							IF HMI_WorkAreaDataPicking[i].NumElementiDaLavorare > 0 THEN 
								NuEstacionesPiking := NuEstacionesPiking + 1 ;	
								PosCavalleteOrdenPikin[i]	:=  e_Tipo_Pallet.CAVALLETTO;  
							END_IF
							BUNDLE_VERT:
								WorkareaState[i].Supporto.Tipologia := e_Tipo_Pallet.BUNDLE;	
							
						 ELSE
								WorkareaState[i].Supporto.Tipologia := e_Tipo_Pallet.CASSA_STANDARD;		   
						 END_CASE
					ELSE
						NumPostazioneDeposito := i; NuEstacionPiking := i;
						
						HMI_WorkAreaDataPicking[NumPostazioneDeposito].NumElementiDaLavorare := RequestPickingListFromHMI[IdxLista].SlabNumber;
						CASE HMI_WorkAreaDataPicking[i].Typology OF
							LEGNO_PIANO,TELAIO_PIANO:
								WorkareaState[i].Supporto.Tipologia := e_Tipo_Pallet.CASSA_STANDARD;
							A_FRAME_VERT:	
								WorkareaState[i].Supporto.Tipologia := e_Tipo_Pallet.CAVALLETTO;
								NuEstacionesPiking := NuEstacionesPiking + 1 ;	
								PosCavalleteOrdenPikin[i]	:=  e_Tipo_Pallet.CAVALLETTO;  	 
							BUNDLE_VERT:
								WorkareaState[i].Supporto.Tipologia := e_Tipo_Pallet.BUNDLE;	
								
							
						 ELSE
								WorkareaState[i].Supporto.Tipologia := e_Tipo_Pallet.CASSA_STANDARD;		   
						 END_CASE
					END_IF

		  
//HMI_NumeroPezziPresentiPostazione[i] := WorkAreaState[i].P -1; //NB:cancellato xckè alla attivazione azzerava il num.pezzi presenti sulle postazioni di prelievo
				END_FOR
	
				IF ElementiDaDepositare[IdxLista] <= HMI_WorkAreaDataPicking[NumPostazioneDeposito].NumElementiDaLavorare THEN
					ActualPickingListFromHMI[IdxLista] 			:= RequestPickingListFromHMI[IdxLista];
					ActualPickingListFromHMI[IdxLista].State 	:= e_StatoWorkOrder.DA_ESEGUIRE;

				ELSE
					HMI_ErroreCalcoloLista := 1;
				END_IF
				Cmd_AttivaLista[IdxLista] 				:= FALSE;
				 
			ELSE
				Cmd_AttivaLista[IdxLista] 				:= FALSE;
				 
			END_IF
{endregion}	

{region "Cotas posicione de trabajo"}

//--------------------------------------------------------------------				
//////// attivazione lista di picking : StatoWorkOrder.DA_ESEGUIRE ///
//--------------------------------------------------------------------				
			IF ActualPickingListFromHMI[IdxLista].State = e_StatoWorkOrder.DA_ESEGUIRE  THEN
				ListaInEsecuzione[IdxLista] := FALSE;
				NumeroListaInEsecuzione := 0;
			
				(* Inserimento sequenza di prelievo dalle postazioni in base al quello che l'operatore ha editato da HMI*)
				ElementiDaDepositare[IdxLista] := 0;
				ElementiElaborati[IdxLista]    := 1;
				NumPostazioneDeposito := 0;
				//FOR i:= 1 TO MAXAREAPRESENT DO
				//	WorkAreaState[i].P := 1;
				//END_FOR		
				
				FOR i:= Iforstart TO Iforend DO//---------- For 1 HMI_WorkAreaDataPicking[i].Destinazione 
					IF HMI_WorkAreaDataPicking[i].Destinazione THEN  //-------> Palet destino
						NumPostazioneDeposito := i;
						HMI_WorkAreaDataPicking[NumPostazioneDeposito].NumElementiDaLavorare 	:= RequestPickingListFromHMI[IdxLista].SlabNumber;
						(*CASE HMI_WorkAreaDataPicking[i].Typology OF     // case Pricipal1*)		 
						CASE HMI_WorkAreaDataPicking[NumPostazioneDeposito].Typology OF     // case Pricipal1	
							(* Se ho un legno in piano *)	 
							LEGNO_PIANO:	
								//WorkAreaState[NumPostazioneDeposito].Supporto.Code 						:= ActualPickingListFromHMI[IdxLista].SupportPianoLegno.Code; 
								WorkAreaState[NumPostazioneDeposito].Supporto.Code 						:= RequestPickingListFromHMIWorkArea[i].SupportPianoLegno.Code; 	   
								//WorkAreaState[NumPostazioneDeposito].Supporto.AltezzaDenteRitenuta 		:= ActualPickingListFromHMI[IdxLista].SupportPianoLegno.DimBaseUtile;
								WorkAreaState[NumPostazioneDeposito].Supporto.AltezzaDenteRitenuta 		:= RequestPickingListFromHMIWorkArea[i].SupportPianoLegno.DimBaseUtile;
								//WorkAreaState[NumPostazioneDeposito].Supporto.DimVertice 				:= ActualPickingListFromHMI[IdxLista].SupportPianoLegno.DimVertice;
								WorkAreaState[NumPostazioneDeposito].Supporto.DimVertice 				:= RequestPickingListFromHMIWorkArea[i].SupportPianoLegno.DimVertice;			   
								//WorkAreaState[NumPostazioneDeposito].Supporto.HMAX 						:= ActualPickingListFromHMI[IdxLista].SupportPianoLegno.HMAX;
							   	WorkAreaState[NumPostazioneDeposito].Supporto.HMAX 						:= RequestPickingListFromHMIWorkArea[i].SupportPianoLegno.HMAX;
								//WorkAreaState[NumPostazioneDeposito].Supporto.Tipologia 				:= e_Tipo_Pallet.CASSA_STANDARD;//ActualPickingListFromHMI.Support.Tipologia;
								WorkAreaState[NumPostazioneDeposito].Supporto.Tipologia 				:= e_Tipo_Pallet.CASSA_STANDARD;//ActualPickingListFromHMI.Support.Tipologia;   
								//WorkAreaState[NumPostazioneDeposito].Supporto.XDim 						:= ActualPickingListFromHMI[IdxLista].SupportPianoLegno.XDim;
								WorkAreaState[NumPostazioneDeposito].Supporto.XDim 						:= RequestPickingListFromHMIWorkArea[i].SupportPianoLegno.XDim;
								//WorkAreaState[NumPostazioneDeposito].Supporto.YDim 						:= ActualPickingListFromHMI[IdxLista].SupportPianoLegno.YDim;
								WorkAreaState[NumPostazioneDeposito].Supporto.YDim 						:= RequestPickingListFromHMIWorkArea[i].SupportPianoLegno.YDim;
								//WorkAreaState[NumPostazioneDeposito].Supporto.ZDim 						:= ActualPickingListFromHMI[IdxLista].SupportPianoLegno.ZDim;
								WorkAreaState[NumPostazioneDeposito].Supporto.ZDim 						:= RequestPickingListFromHMIWorkArea[i].SupportPianoLegno.ZDim;
								WorkAreaOffset[NumPostazioneDeposito].Y 								:= OFFSET_POSTAZIONE_LEGNO + ActualPickingListFromHMI[IdxLista].SupportPianoLegno.YDim/2;//ATTENZIONE!!! per poter lavorare in centro con i supporti pari, questa misura è la distanza tra il riscontro bundle verticale e il centro postazione PARI
								
								WorkAreaProductionList[NumPostazioneDeposito].Support 				:= WorkAreaState[NumPostazioneDeposito].Supporto;
								
								FOR j:= Iforstart TO Iforend DO
									IF NOT HMI_WorkAreaDataPicking[j].Destinazione THEN
										IF HMI_WorkAreaDataPicking[j].NumElementiDaLavorare >= 1 THEN
											ElementiDaDepositare[IdxLista] := ElementiElaborati[IdxLista] + HMI_WorkAreaDataPicking[j].NumElementiDaLavorare;
											FOR k := ElementiElaborati[IdxLista] TO ElementiDaDepositare[IdxLista]-1 DO	
												WorkAreaProductionList[NumPostazioneDeposito].PElementList[k].WA_PRELIEVO := j;
												WorkAreaProductionList[NumPostazioneDeposito].PElementList[k].WA_DEPOSITO := i;	
												// Se van Añadiendo los Diferentes Espesores de la receta del piking ######################################
												HMi_DimensionesPiezasWorkAreaDeposito[K] := RequestPickingListFromHMIWorkArea[j].SlabDimension ;
												//########################################################################################################
												ElementiElaborati[IdxLista] := ElementiElaborati[IdxLista]+1; 
											END_FOR
											CASE HMI_WorkAreaDataPicking[j].Typology OF 
												(* Se ho una cassa pianale in legno *)
												LEGNO_PIANO:
													WorkAreaState[j].Supporto.Code 					:= RequestPickingListFromHMIWorkArea[j].SupportPianoLegno.Code;
													WorkAreaState[j].Supporto.DimBaseUtile		 	:= RequestPickingListFromHMIWorkArea[j].SupportPianoLegno.DimBaseUtile;
													WorkAreaState[j].Supporto.AltezzaDenteRitenuta 	:= RequestPickingListFromHMIWorkArea[j].SupportPianoLegno.ZDim+20;
													WorkAreaState[j].Supporto.DimVertice 			:= RequestPickingListFromHMIWorkArea[j].SupportPianoLegno.DimVertice;
													WorkAreaState[j].Supporto.HMAX 					:= RequestPickingListFromHMIWorkArea[j].SupportPianoLegno.HMAX;
													WorkAreaState[j].Supporto.Tipologia 			:= e_Tipo_Pallet.CASSA_STANDARD;//ActualPickingListFromHMI[1].Support.Tipologia;
													WorkAreaState[j].Supporto.XDim 					:= RequestPickingListFromHMIWorkArea[j].SupportPianoLegno.XDim;
													WorkAreaState[j].Supporto.YDim 					:= RequestPickingListFromHMIWorkArea[j].SupportPianoLegno.YDim;
													WorkAreaState[j].Supporto.ZDim 					:= RequestPickingListFromHMIWorkArea[j].SupportPianoLegno.ZDim;
													WorkAreaOffset[j].Y 							:= OFFSET_POSTAZIONE_LEGNO + ActualPickingListFromHMI[IdxLista].SupportPianoLegno.YDim/2;//ATTENZIONE!!! per poter lavorare in centro con i supporti pari, questa misura è la distanza tra il riscontro bundle verticale e il centro postazione PARI
													
																   
												(* Se ho una cassa pianale in ferro su supporto *)
												TELAIO_PIANO:
													WorkAreaState[j].Supporto.Code 					:= RequestPickingListFromHMIWorkArea[j].SupportPianoFerro.Code;
													WorkAreaState[j].Supporto.DimBaseUtile		 	:= RequestPickingListFromHMIWorkArea[j].SupportPianoFerro.DimBaseUtile;
													WorkAreaState[j].Supporto.AltezzaDenteRitenuta 	:= RequestPickingListFromHMIWorkArea[j].SupportPianoFerro.ZDim+20;
													WorkAreaState[j].Supporto.DimVertice 			:= RequestPickingListFromHMIWorkArea[j].SupportPianoFerro.DimVertice;
													WorkAreaState[j].Supporto.HMAX 					:= RequestPickingListFromHMIWorkArea[j].SupportPianoFerro.HMAX;
													WorkAreaState[j].Supporto.Tipologia 			:=  e_Tipo_Pallet.CASSA_STANDARD;//ActualPickingListFromHMI[1].Support.Tipologia;
													WorkAreaState[j].Supporto.XDim 					:= RequestPickingListFromHMIWorkArea[j].SupportPianoFerro.XDim;
													WorkAreaState[j].Supporto.YDim 					:= RequestPickingListFromHMIWorkArea[j].SupportPianoFerro.YDim;
													WorkAreaState[j].Supporto.ZDim 					:= RequestPickingListFromHMIWorkArea[j].SupportPianoFerro.ZDim;
													WorkAreaOffset[j].Y 							:= OFFSET_POSTAZIONE_TELAIO - ActualPickingListFromHMI[IdxLista].SupportPianoFerro.YDim/2;//ATTENZIONE!!! per poter lavorare in centro con i supporti pari, questa misura è la distanza tra il riscontro bundle verticale e il centro postazione PARI
												(* Se ho un bundle *)
												BUNDLE_VERT:
													//WorkAreaState[j].P := ElementiDaDepositare;
													WorkAreaState[j].Supporto.Code 					:= RequestPickingListFromHMIWorkArea[j].SupportVertBundle.Code;
													WorkAreaState[j].Supporto.DimBaseUtile		 	:= RequestPickingListFromHMIWorkArea[j].SupportVertBundle.DimBaseUtile;
													WorkAreaState[j].Supporto.AltezzaDenteRitenuta 	:= RequestPickingListFromHMIWorkArea[j].SupportVertBundle.ZDim+20;
													WorkAreaState[j].Supporto.DimVertice 			:= RequestPickingListFromHMIWorkArea[j].SupportVertBundle.DimVertice;
													WorkAreaState[j].Supporto.HMAX 					:= RequestPickingListFromHMIWorkArea[j].SupportVertBundle.HMAX;
													WorkAreaState[j].Supporto.Tipologia 			:= e_Tipo_Pallet.BUNDLE;//ActualPickingListFromHMI.SupportVert.Tipologia;
													WorkAreaState[j].Supporto.XDim 					:= RequestPickingListFromHMIWorkArea[j].SupportVertBundle.XDim;
													WorkAreaState[j].Supporto.YDim 					:= RequestPickingListFromHMIWorkArea[j].SupportVertBundle.YDim;
													WorkAreaState[j].Supporto.ZDim 					:= RequestPickingListFromHMIWorkArea[j].SupportVertBundle.ZDim;
													WorkAreaState[j].Supporto.ZDim_Ext1        		:= WorkAreaState[j].Supporto.ZDim + 20;
													WorkAreaState[j].Supporto.TipoPianoAppoggio 	:= 1;                      
													WorkAreaState[j].Supporto.AltezzaDenteRitenuta	:= 20; 
													WorkAreaState[j].Supporto.LatoDeposito 			:= 180;    
													//Lo que HABIA	
													//WorkAreaOffset[j].Y 							:= HMI_OffsetDepositoLastra.Y180 ;
													//Mod 25/&/2025	  
													WorkAreaOffset[NumPostazioneDeposito].Y 		:= RequestPickingListFromHMIWorkArea[j].SupportVertBundle.YDim - RequestPickingListFromHMIWorkArea[j].SupportVertBundle.DimBaseUtile -40 ;			
												(* Se ho un A_Frame *)	  
												A_FRAME_VERT:  						
													//WorkAreaState[j].P := ElementiDaDepositare;
													WorkAreaState[j].Supporto.Code 					:= ActualPickingListFromHMI[IdxLista].SupportVertCav.Code;
													WorkAreaState[j].Supporto.DimBaseUtile		 	:= RequestPickingListFromHMIWorkArea[j].SupportVertCav.DimBaseUtile;
													WorkAreaState[j].Supporto.AltezzaDenteRitenuta 	:= RequestPickingListFromHMIWorkArea[j].SupportVertCav.ZDim+20;
													WorkAreaState[j].Supporto.DimVertice 			:= RequestPickingListFromHMIWorkArea[j].SupportVertCav.DimVertice;
													WorkAreaState[j].Supporto.HMAX 					:= RequestPickingListFromHMIWorkArea[j].SupportVertCav.HMAX;
													WorkAreaState[j].Supporto.Tipologia 			:= CAVALLETTO;//ActualPickingListFromHMI.SupportVertCav.Tipologia;
													WorkAreaState[j].Supporto.XDim 					:= RequestPickingListFromHMIWorkArea[j].SupportVertCav.XDim;
													WorkAreaState[j].Supporto.YDim 					:= RequestPickingListFromHMIWorkArea[j].SupportVertCav.YDim;
													WorkAreaState[j].Supporto.ZDim 					:= RequestPickingListFromHMIWorkArea[j].SupportVertCav.ZDim;
													WorkAreaState[j].Supporto.ZDim_Ext1        		:= WorkAreaState[j].Supporto.ZDim + 20;	
													WorkAreaState[j].Supporto.TipoPianoAppoggio 	:= 1;                      
													WorkAreaState[j].Supporto.AltezzaDenteRitenuta	:= 15;     	
													WorkAreaOffset[j].Y 							:= OFFSET_POSTAZIONE_LEGNO + ActualPickingListFromHMI[IdxLista].SupportVertCav.YDim/2;//ATTENZIONE!!! per poter lavorare in centro con i supporti pari, questa misura è la distanza tra il riscontro bundle verticale e il centro postazione PARI
											   		CoordenadaPasillo0_Y 							:= WorkArea[j].Y +  WorkAreaOffset[j].Y  - Dimensioni_Pinza.Spessore - INGOMBRO_RISCONTRO_BUNDLE - WorkAreaState[j].Supporto.YDim /2 ;
													CoordenadaPasillo180_Y 							:= WorkArea[j].Y + WorkAreaState[j].Supporto.YDim /2 + WorkAreaOffset[j].Y  + Dimensioni_Pinza.Spessore + INGOMBRO_RISCONTRO_FRAME  ;	
											END_CASE	
											WorkAreaProductionList[j].Support := WorkAreaState[j].Supporto; 
										END_IF
									END_IF     
									TFClearApprendimento(ADR(WorkAreaState[j].Apprendimento));//Azzeramento apprendimento 
								END_FOR
								EXIT; 
							(* Se ho un telaio in piano *)	 
							TELAIO_PIANO:	
								WorkAreaState[NumPostazioneDeposito].Supporto.Code 						:= ActualPickingListFromHMI[IdxLista].SupportPianoFerro.Code;
								WorkAreaState[NumPostazioneDeposito].Supporto.AltezzaDenteRitenuta 		:= RequestPickingListFromHMIWorkArea[j].SupportPianoFerro.DimBaseUtile;
								WorkAreaState[NumPostazioneDeposito].Supporto.DimVertice 				:= RequestPickingListFromHMIWorkArea[j].SupportPianoFerro.DimVertice;
								WorkAreaState[NumPostazioneDeposito].Supporto.HMAX 						:= RequestPickingListFromHMIWorkArea[j].SupportPianoFerro.HMAX;
								WorkAreaState[NumPostazioneDeposito].Supporto.Tipologia 				:= CASSA_STANDARD;//ActualPickingListFromHMI.Support.Tipologia;
								WorkAreaState[NumPostazioneDeposito].Supporto.XDim 						:= RequestPickingListFromHMIWorkArea[j].SupportPianoFerro.XDim;
								WorkAreaState[NumPostazioneDeposito].Supporto.YDim 						:= RequestPickingListFromHMIWorkArea[j].SupportPianoFerro.YDim;
								WorkAreaState[NumPostazioneDeposito].Supporto.ZDim 						:= RequestPickingListFromHMIWorkArea[j].SupportPianoFerro.ZDim;
								WorkAreaOffset[NumPostazioneDeposito].Y 								:= OFFSET_POSTAZIONE_TELAIO - ActualPickingListFromHMI[IdxLista].SupportPianoFerro.YDim/2;//ATTENZIONE!!! per poter lavorare in centro con i supporti pari, questa misura è la distanza tra il riscontro bundle verticale e il centro postazione PARI
								
								WorkAreaProductionList[NumPostazioneDeposito].Support := WorkAreaState[NumPostazioneDeposito].Supporto;
							
								
								FOR j:= Iforstart TO Iforend DO
									IF NOT HMI_WorkAreaDataPicking[j].Destinazione THEN
										IF HMI_WorkAreaDataPicking[j].NumElementiDaLavorare >= 1 THEN
											ElementiDaDepositare[IdxLista] := ElementiElaborati[IdxLista] + HMI_WorkAreaDataPicking[j].NumElementiDaLavorare;
											FOR k := ElementiElaborati[IdxLista] TO ElementiDaDepositare[IdxLista]-1 DO	
												WorkAreaProductionList[NumPostazioneDeposito].PElementList[k].WA_PRELIEVO := j;
												WorkAreaProductionList[NumPostazioneDeposito].PElementList[k].WA_DEPOSITO := i;	
												// Se van Añadiendo los Diferentes Espesores de la receta del piking ######################################
												HMi_DimensionesPiezasWorkAreaDeposito[K] := RequestPickingListFromHMIWorkArea[j].SlabDimension ;
												//########################################################################################################
												ElementiElaborati[IdxLista] := ElementiElaborati[IdxLista]+1; 
											END_FOR
											CASE HMI_WorkAreaDataPicking[j].Typology OF 
												(* Se ho una cassa pianale in legno *)
												LEGNO_PIANO:
													WorkAreaState[j].Supporto.Code 					:= ActualPickingListFromHMI[IdxLista].SupportPianoLegno.Code;
													WorkAreaState[j].Supporto.DimBaseUtile		 	:= RequestPickingListFromHMIWorkArea[j].SupportPianoLegno.DimBaseUtile;
													WorkAreaState[j].Supporto.AltezzaDenteRitenuta 	:= RequestPickingListFromHMIWorkArea[j].SupportPianoLegno.ZDim+20;
													WorkAreaState[j].Supporto.DimVertice 			:= RequestPickingListFromHMIWorkArea[j].SupportPianoLegno.DimVertice;
													WorkAreaState[j].Supporto.HMAX 					:= RequestPickingListFromHMIWorkArea[j].SupportPianoLegno.HMAX;
													WorkAreaState[j].Supporto.Tipologia 			:=  e_Tipo_Pallet.CASSA_STANDARD;//ActualPickingListFromHMI[1].Support.Tipologia;
													WorkAreaState[j].Supporto.XDim 					:= RequestPickingListFromHMIWorkArea[j].SupportPianoLegno.XDim;
													WorkAreaState[j].Supporto.YDim 					:= RequestPickingListFromHMIWorkArea[j].SupportPianoLegno.YDim;
													WorkAreaState[j].Supporto.ZDim 					:= RequestPickingListFromHMIWorkArea[j].SupportPianoLegno.ZDim;
													WorkAreaOffset[j].Y 							:= OFFSET_POSTAZIONE_LEGNO + ActualPickingListFromHMI[IdxLista].SupportPianoLegno.YDim/2;//ATTENZIONE!!! per poter lavorare in centro con i supporti pari, questa misura è la distanza tra il riscontro bundle verticale e il centro postazione PARI
												(* Se ho una cassa pianale in ferro su supporto *)
												TELAIO_PIANO:
													WorkAreaState[j].Supporto.Code 					:= ActualPickingListFromHMI[IdxLista].SupportPianoFerro.Code;
													WorkAreaState[j].Supporto.DimBaseUtile		 	:= RequestPickingListFromHMIWorkArea[j].SupportPianoFerro.DimBaseUtile;
													WorkAreaState[j].Supporto.AltezzaDenteRitenuta 	:= RequestPickingListFromHMIWorkArea[j].SupportPianoFerro.ZDim+20;
													WorkAreaState[j].Supporto.DimVertice 			:= RequestPickingListFromHMIWorkArea[j].SupportPianoFerro.DimVertice;
													WorkAreaState[j].Supporto.HMAX 					:= RequestPickingListFromHMIWorkArea[j].SupportPianoFerro.HMAX;
													WorkAreaState[j].Supporto.Tipologia 			:=  e_Tipo_Pallet.CASSA_STANDARD;//ActualPickingListFromHMI[1].Support.Tipologia;
													WorkAreaState[j].Supporto.XDim 					:= RequestPickingListFromHMIWorkArea[j].SupportPianoFerro.XDim;
													WorkAreaState[j].Supporto.YDim 					:= RequestPickingListFromHMIWorkArea[j].SupportPianoFerro.YDim;
													WorkAreaState[j].Supporto.ZDim 					:= RequestPickingListFromHMIWorkArea[j].SupportPianoFerro.ZDim;
													WorkAreaOffset[j].Y 							:= OFFSET_POSTAZIONE_TELAIO - ActualPickingListFromHMI[IdxLista].SupportPianoFerro.YDim/2;//ATTENZIONE!!! per poter lavorare in centro con i supporti pari, questa misura è la distanza tra il riscontro bundle verticale e il centro postazione PARI
												(* Se ho un bundle *)
												BUNDLE_VERT:
													//WorkAreaState[j].P := ElementiDaDepositare;
													WorkAreaState[j].Supporto.Code 					:= RequestPickingListFromHMIWorkArea[j].SupportVertBundle.Code;
													WorkAreaState[j].Supporto.DimBaseUtile		 	:= RequestPickingListFromHMIWorkArea[j].SupportVertBundle.DimBaseUtile;
													WorkAreaState[j].Supporto.AltezzaDenteRitenuta 	:= RequestPickingListFromHMIWorkArea[j].SupportVertBundle.ZDim+20;
													WorkAreaState[j].Supporto.DimVertice 			:= RequestPickingListFromHMIWorkArea[j].SupportVertBundle.DimVertice;
													WorkAreaState[j].Supporto.HMAX 					:= RequestPickingListFromHMIWorkArea[j].SupportVertBundle.HMAX;
													WorkAreaState[j].Supporto.Tipologia 			:= e_Tipo_Pallet.BUNDLE;//ActualPickingListFromHMI.SupportVertBundle.Tipologia;
													WorkAreaState[j].Supporto.XDim 					:= RequestPickingListFromHMIWorkArea[j].SupportVertBundle.XDim;
													WorkAreaState[j].Supporto.YDim 					:= RequestPickingListFromHMIWorkArea[j].SupportVertBundle.YDim;
													WorkAreaState[j].Supporto.ZDim 					:= RequestPickingListFromHMIWorkArea[j].SupportVertBundle.ZDim;
													WorkAreaState[j].Supporto.ZDim_Ext1        		:= WorkAreaState[j].Supporto.ZDim + 20;
													WorkAreaState[j].Supporto.TipoPianoAppoggio 	:= 1;                      
													WorkAreaState[j].Supporto.AltezzaDenteRitenuta	:= 20; 
													WorkAreaState[j].Supporto.LatoDeposito 			:= 180;   	
													  
													WorkAreaOffset[j].Y 		:= 0 ;	
													//Mod 25/&/2025	  
													//WorkAreaOffset[j].Y 		:= ActualPickingListFromHMI[IdxLista].SupportVertBundle.YDim-ActualPickingListFromHMI[IdxLista].SupportVertBundle.DimBaseUtile -40;				
												(* Se ho un A_Frame *)	  
												A_FRAME_VERT:  						
													//WorkAreaState[j].P := ElementiDaDepositare;
													WorkAreaState[j].Supporto.Code 					:= ActualPickingListFromHMI[IdxLista].SupportVertCav.Code;
													WorkAreaState[j].Supporto.DimBaseUtile		 	:= RequestPickingListFromHMIWorkArea[j].SupportVertCav.DimBaseUtile;
													WorkAreaState[j].Supporto.AltezzaDenteRitenuta 	:= RequestPickingListFromHMIWorkArea[j].SupportVertCav.ZDim+20;
													WorkAreaState[j].Supporto.DimVertice 			:= RequestPickingListFromHMIWorkArea[j].SupportVertCav.DimVertice;
													WorkAreaState[j].Supporto.HMAX 					:= RequestPickingListFromHMIWorkArea[j].SupportVertcav.HMAX;
													WorkAreaState[j].Supporto.Tipologia 			:= CAVALLETTO;//ActualPickingListFromHMI.SupportVert.Tipologia;
													WorkAreaState[j].Supporto.XDim 					:= RequestPickingListFromHMIWorkArea[j].SupportVertCav.XDim;
													WorkAreaState[j].Supporto.YDim 					:= RequestPickingListFromHMIWorkArea[j].SupportVertCav.YDim;
													WorkAreaState[j].Supporto.ZDim 					:= RequestPickingListFromHMIWorkArea[j].SupportVertCav.ZDim;
													WorkAreaState[j].Supporto.ZDim_Ext1        		:= WorkAreaState[j].Supporto.ZDim + 20;	
													WorkAreaState[j].Supporto.TipoPianoAppoggio 	:= 1;                      
													WorkAreaState[j].Supporto.AltezzaDenteRitenuta	:= 15; 	
													WorkAreaOffset[j].Y 							:= OFFSET_POSTAZIONE_LEGNO + ActualPickingListFromHMI[IdxLista].SupportVertCav.YDim/2;//ATTENZIONE!!! per poter lavorare in centro con i supporti pari, questa misura è la distanza tra il riscontro bundle verticale e il centro postazione PARI
											   		CoordenadaPasillo0_Y 							:= WorkArea[j].Y +  WorkAreaOffset[j].Y  - Dimensioni_Pinza.Spessore - INGOMBRO_RISCONTRO_BUNDLE - WorkAreaState[j].Supporto.YDim /2 ;
													CoordenadaPasillo180_Y 							:= WorkArea[j].Y + WorkAreaState[j].Supporto.YDim /2 + WorkAreaOffset[j].Y  + Dimensioni_Pinza.Spessore + INGOMBRO_RISCONTRO_FRAME  ;	
											END_CASE	
											WorkAreaProductionList[j].Support := WorkAreaState[j].Supporto; 
										END_IF
									END_IF     
									TFClearApprendimento(ADR(WorkAreaState[j].Apprendimento));//Azzeramento apprendimento 
								END_FOR
								EXIT; 
							(* Se ho un bundle *)
							BUNDLE_VERT:
								
								//Se ho deposito verticale su bundle
								WorkAreaState[NumPostazioneDeposito].Supporto.Code 						:= ActualPickingListFromHMI[IdxLista].SupportVertBundle.Code;
								WorkAreaState[NumPostazioneDeposito].Supporto.DimBaseUtile		 		:= RequestPickingListFromHMIWorkArea[j].SupportVertBundle.DimBaseUtile;
								WorkAreaState[NumPostazioneDeposito].Supporto.DimVertice 				:= RequestPickingListFromHMIWorkArea[j].SupportVertBundle.DimVertice;
								WorkAreaState[NumPostazioneDeposito].Supporto.HMAX 						:= RequestPickingListFromHMIWorkArea[j].SupportVertBundle.HMAX;
								WorkAreaState[NumPostazioneDeposito].Supporto.Tipologia 				:= e_Tipo_Pallet.BUNDLE;
								WorkAreaState[NumPostazioneDeposito].Supporto.XDim 						:= RequestPickingListFromHMIWorkArea[j].SupportVertBundle.XDim;
								WorkAreaState[NumPostazioneDeposito].Supporto.YDim 						:= RequestPickingListFromHMIWorkArea[j].SupportVertBundle.YDim;
								WorkAreaState[NumPostazioneDeposito].Supporto.ZDim 						:= RequestPickingListFromHMIWorkArea[j].SupportVertBundle.ZDim;
								WorkAreaState[NumPostazioneDeposito].Supporto.TipoPianoAppoggio 		:= 1;                      
								WorkAreaState[NumPostazioneDeposito].Supporto.AltezzaDenteRitenuta		:= 20; 
								WorkAreaState[NumPostazioneDeposito].Supporto.LatoDeposito 				:= 180; 
											   
								WorkAreaProductionList[NumPostazioneDeposito].Support 					:= WorkAreaState[NumPostazioneDeposito].Supporto;
								
								FOR j:= Iforstart TO Iforend DO
									IF NOT HMI_WorkAreaDataPicking[j].Destinazione THEN
										IF HMI_WorkAreaDataPicking[j].NumElementiDaLavorare >= 1 THEN
											ElementiDaDepositare[IdxLista] := ElementiElaborati[IdxLista] + HMI_WorkAreaDataPicking[j].NumElementiDaLavorare;
											FOR k := ElementiElaborati[IdxLista] TO ElementiDaDepositare[IdxLista]-1 DO	
												WorkAreaProductionList[NumPostazioneDeposito].PElementList[k].WA_PRELIEVO := j;
												WorkAreaProductionList[NumPostazioneDeposito].PElementList[k].WA_DEPOSITO := i;	
												// Se van Añadiendo los Diferentes Espesores de la receta del piking ######################################
												HMi_DimensionesPiezasWorkAreaDeposito[K] := RequestPickingListFromHMIWorkArea[j].SlabDimension ;
												//########################################################################################################
												ElementiElaborati[IdxLista] := ElementiElaborati[IdxLista]+1; 
											END_FOR
											CASE HMI_WorkAreaDataPicking[j].Typology OF 
												(* Se ho una cassa pianale in legno *)
												LEGNO_PIANO:
													WorkAreaState[j].Supporto.Code 					:= ActualPickingListFromHMI[IdxLista].SupportPianoLegno.Code;
													WorkAreaState[j].Supporto.DimBaseUtile		 	:= RequestPickingListFromHMIWorkArea[j].SupportPianoLegno.DimBaseUtile;
													WorkAreaState[j].Supporto.AltezzaDenteRitenuta 	:= RequestPickingListFromHMIWorkArea[j].SupportPianoLegno.ZDim+20;
													WorkAreaState[j].Supporto.DimVertice 			:= RequestPickingListFromHMIWorkArea[j].SupportPianoLegno.DimVertice;
													WorkAreaState[j].Supporto.HMAX 					:= RequestPickingListFromHMIWorkArea[j].SupportPianoLegno.HMAX;
													WorkAreaState[j].Supporto.Tipologia 			:=  e_Tipo_Pallet.CASSA_STANDARD;//ActualPickingListFromHMI[1].Support.Tipologia;
													WorkAreaState[j].Supporto.XDim 					:= RequestPickingListFromHMIWorkArea[j].SupportPianoLegno.XDim;
													WorkAreaState[j].Supporto.YDim 					:= RequestPickingListFromHMIWorkArea[j].SupportPianoLegno.YDim;
													WorkAreaState[j].Supporto.ZDim 					:= RequestPickingListFromHMIWorkArea[j].SupportPianoLegno.ZDim;
													WorkAreaOffset[j].Y 							:= OFFSET_POSTAZIONE_LEGNO + ActualPickingListFromHMI[IdxLista].SupportPianoLegno.YDim/2;//ATTENZIONE!!! per poter lavorare in centro con i supporti pari, questa misura è la distanza tra il riscontro bundle verticale e il centro postazione PARI
												(* Se ho una cassa pianale in ferro su supporto *)
												TELAIO_PIANO:
													WorkAreaState[j].Supporto.Code 					:= ActualPickingListFromHMI[IdxLista].SupportPianoFerro.Code;
													WorkAreaState[j].Supporto.DimBaseUtile		 	:= RequestPickingListFromHMIWorkArea[j].SupportPianoFerro.DimBaseUtile;
													WorkAreaState[j].Supporto.AltezzaDenteRitenuta 	:= RequestPickingListFromHMIWorkArea[j].SupportPianoFerro.ZDim+20;
													WorkAreaState[j].Supporto.DimVertice 			:= RequestPickingListFromHMIWorkArea[j].SupportPianoFerro.DimVertice;
													WorkAreaState[j].Supporto.HMAX 					:= RequestPickingListFromHMIWorkArea[j].SupportPianoFerro.HMAX;
													WorkAreaState[j].Supporto.Tipologia 			:=  e_Tipo_Pallet.CASSA_STANDARD;//ActualPickingListFromHMI[1].Support.Tipologia;
													WorkAreaState[j].Supporto.XDim 					:= RequestPickingListFromHMIWorkArea[j].SupportPianoFerro.XDim;
													WorkAreaState[j].Supporto.YDim 					:= RequestPickingListFromHMIWorkArea[j].SupportPianoFerro.YDim;
													WorkAreaState[j].Supporto.ZDim 					:= RequestPickingListFromHMIWorkArea[j].SupportPianoFerro.ZDim;
													WorkAreaOffset[j].Y 							:= OFFSET_POSTAZIONE_TELAIO - ActualPickingListFromHMI[IdxLista].SupportPianoFerro.YDim/2;//ATTENZIONE!!! per poter lavorare in centro con i supporti pari, questa misura è la distanza tra il riscontro bundle verticale e il centro postazione PARI
												(* Se ho un bundle *)
												BUNDLE_VERT:
													//WorkAreaState[j].P := ElementiDaDepositare;
													WorkAreaState[j].Supporto.Code 					:= ActualPickingListFromHMI[IdxLista].SupportVertBundle.Code;
													WorkAreaState[j].Supporto.DimBaseUtile		 	:= RequestPickingListFromHMIWorkArea[j].SupportVertBundle.DimBaseUtile;
													WorkAreaState[j].Supporto.AltezzaDenteRitenuta 	:= RequestPickingListFromHMIWorkArea[j].SupportVertBundle.ZDim+20;
													WorkAreaState[j].Supporto.DimVertice 			:= RequestPickingListFromHMIWorkArea[j].SupportVertBundle.DimVertice;
													WorkAreaState[j].Supporto.HMAX 					:= RequestPickingListFromHMIWorkArea[j].SupportVertBundle.HMAX;
													WorkAreaState[j].Supporto.Tipologia 			:= e_Tipo_Pallet.BUNDLE;//ActualPickingListFromHMI.SupportVert.Tipologia;
													WorkAreaState[j].Supporto.XDim 					:= RequestPickingListFromHMIWorkArea[j].SupportVertBundle.XDim;
													WorkAreaState[j].Supporto.YDim 					:= RequestPickingListFromHMIWorkArea[j].SupportVertBundle.YDim;
													WorkAreaState[j].Supporto.ZDim 					:= RequestPickingListFromHMIWorkArea[j].SupportVertBundle.ZDim;
													WorkAreaState[j].Supporto.ZDim_Ext1        		:= WorkAreaState[j].Supporto.ZDim + 20;	
													// **Lo Que Habia	
													WorkAreaOffset[j].Y 							:= 0;
													//Mod 25/&/2025	  
													//WorkAreaOffset[j].Y 		:= ActualPickingListFromHMI[IdxLista].SupportVertBundle.YDim-ActualPickingListFromHMI[IdxLista].SupportVertBundle.DimBaseUtile -40;	
			
												(* Se ho un A_Frame *)	  
												A_FRAME_VERT:  						
													//WorkAreaState[j].P := ElementiDaDepositare;
													WorkAreaState[j].Supporto.Code 					:= ActualPickingListFromHMI[IdxLista].SupportVertCav.Code;
													WorkAreaState[j].Supporto.DimBaseUtile		 	:= RequestPickingListFromHMIWorkArea[j].SupportVertCav.DimBaseUtile;
													WorkAreaState[j].Supporto.AltezzaDenteRitenuta 	:= RequestPickingListFromHMIWorkArea[j].SupportVertCav.ZDim+20;
													WorkAreaState[j].Supporto.DimVertice 			:= RequestPickingListFromHMIWorkArea[j].SupportVertCav.DimVertice;
													WorkAreaState[j].Supporto.HMAX 					:= RequestPickingListFromHMIWorkArea[j].SupportVertCav.HMAX;
													WorkAreaState[j].Supporto.Tipologia 			:= CAVALLETTO;//ActualPickingListFromHMI.SupportVert.Tipologia;
													WorkAreaState[j].Supporto.XDim 					:= RequestPickingListFromHMIWorkArea[j].SupportVertCav.XDim;
													WorkAreaState[j].Supporto.YDim 					:= RequestPickingListFromHMIWorkArea[j].SupportVertCav.YDim;
													WorkAreaState[j].Supporto.ZDim 					:= RequestPickingListFromHMIWorkArea[j].SupportVertCav.ZDim;
													WorkAreaState[j].Supporto.ZDim_Ext1        		:= WorkAreaState[j].Supporto.ZDim + 20;	
													WorkAreaState[j].Supporto.TipoPianoAppoggio 	:= 1;                      
													WorkAreaState[j].Supporto.AltezzaDenteRitenuta	:= 15; 	
													WorkAreaOffset[j].Y 							:= OFFSET_POSTAZIONE_LEGNO + ActualPickingListFromHMI[IdxLista].SupportVertCav.YDim/2;//ATTENZIONE!!! per poter lavorare in centro con i supporti pari, questa misura è la distanza tra il riscontro bundle verticale e il centro postazione PARI
													CoordenadaPasillo0_Y 							:= WorkArea[j].Y +  WorkAreaOffset[j].Y  - Dimensioni_Pinza.Spessore - INGOMBRO_RISCONTRO_BUNDLE - WorkAreaState[j].Supporto.YDim /2 ;
													CoordenadaPasillo180_Y 							:= WorkArea[j].Y + WorkAreaState[j].Supporto.YDim /2 + WorkAreaOffset[j].Y  + Dimensioni_Pinza.Spessore + INGOMBRO_RISCONTRO_FRAME  ;		  
											END_CASE
											//WorkAreaProductionList[j].Support := HMI_Formatura.HMI_Forming_Supporto;		  
											WorkAreaProductionList[j].Support := WorkAreaState[j].Supporto;
										END_IF
									END_IF
									TFClearApprendimento(ADR(WorkAreaState[j].Apprendimento));//Azzeramento apprendimento
								END_FOR
								EXIT; 
							(* Se ho un A_Frame *)	
							A_FRAME_VERT:
								WorkAreaState[NumPostazioneDeposito].Supporto.Code 						:= ActualPickingListFromHMI[IdxLista].SupportVertCav.Code;
								WorkAreaState[NumPostazioneDeposito].Supporto.DimBaseUtile		 		:= RequestPickingListFromHMIWorkArea[j].SupportVertCav.DimBaseUtile;
								WorkAreaState[NumPostazioneDeposito].Supporto.DimVertice 				:= RequestPickingListFromHMIWorkArea[j].SupportVertCav.DimVertice;
								WorkAreaState[NumPostazioneDeposito].Supporto.HMAX 						:= RequestPickingListFromHMIWorkArea[j].SupportVertCav.HMAX;
								WorkAreaState[NumPostazioneDeposito].Supporto.Tipologia 				:= e_Tipo_Pallet.CAVALLETTO;//ActualPickingListFromHMI.SupportVertBundle.Tipologia;
								WorkAreaState[NumPostazioneDeposito].Supporto.XDim 						:= RequestPickingListFromHMIWorkArea[j].SupportVertCav.XDim;
								WorkAreaState[NumPostazioneDeposito].Supporto.YDim 						:= RequestPickingListFromHMIWorkArea[j].SupportVertCav.YDim;
								WorkAreaState[NumPostazioneDeposito].Supporto.ZDim 						:= RequestPickingListFromHMIWorkArea[j].SupportVertCav.ZDim;
								WorkAreaState[NumPostazioneDeposito].Supporto.TipoPianoAppoggio 		:= 1;                      
								WorkAreaState[NumPostazioneDeposito].Supporto.AltezzaDenteRitenuta		:= 15; 
								//WorkAreaOffset[NumPostazioneDeposito].Y 								:= OFFSET_POSTAZIONE_LEGNO (*- ActualPickingListFromHMI[IdxLista].SupportPianoFerro.YDim/2*);
								WorkAreaOffset[NumPostazioneDeposito].Y 								:= OFFSET_POSTAZIONE_LEGNO + ActualPickingListFromHMI[IdxLista].SupportVertCav.YDim/2;	
								
								WorkAreaProductionList[NumPostazioneDeposito].Support 				:= WorkAreaState[NumPostazioneDeposito].Supporto; 
								
								FOR j:= Iforstart TO Iforend DO
									IF NOT HMI_WorkAreaDataPicking[j].Destinazione THEN
										IF HMI_WorkAreaDataPicking[j].NumElementiDaLavorare >= 1 THEN
											ElementiDaDepositare[IdxLista] := ElementiElaborati[IdxLista] + HMI_WorkAreaDataPicking[j].NumElementiDaLavorare;
											FOR k := ElementiElaborati[IdxLista] TO ElementiDaDepositare[IdxLista]-1 DO	
												WorkAreaProductionList[NumPostazioneDeposito].PElementList[k].WA_PRELIEVO := j;
												WorkAreaProductionList[NumPostazioneDeposito].PElementList[k].WA_DEPOSITO := i;	
												// Se van Añadiendo los Diferentes Espesores de la receta del piking ######################################
												HMi_DimensionesPiezasWorkAreaDeposito[K] := RequestPickingListFromHMIWorkArea[j].SlabDimension ;
												//########################################################################################################
												ElementiElaborati[IdxLista] := ElementiElaborati[IdxLista]+1; 
											END_FOR
											CASE HMI_WorkAreaDataPicking[j].Typology OF 
												(* Se ho una cassa pianale in legno *)
												LEGNO_PIANO:
													WorkAreaState[j].Supporto.Code 					:= ActualPickingListFromHMI[IdxLista].SupportPianoLegno.Code;
													WorkAreaState[j].Supporto.DimBaseUtile		 	:= RequestPickingListFromHMIWorkArea[j].SupportPianoLegno.DimBaseUtile;
													WorkAreaState[j].Supporto.AltezzaDenteRitenuta 	:= RequestPickingListFromHMIWorkArea[j].SupportPianoLegno.ZDim+20;
													WorkAreaState[j].Supporto.DimVertice 			:= RequestPickingListFromHMIWorkArea[j].SupportPianoLegno.DimVertice;
													WorkAreaState[j].Supporto.HMAX 					:= RequestPickingListFromHMIWorkArea[j].SupportPianoLegno.HMAX;
													WorkAreaState[j].Supporto.Tipologia 			:=  e_Tipo_Pallet.CASSA_STANDARD;//ActualPickingListFromHMI[1].Support.Tipologia;
													WorkAreaState[j].Supporto.XDim 					:= RequestPickingListFromHMIWorkArea[j].SupportPianoLegno.XDim;
													WorkAreaState[j].Supporto.YDim 					:= RequestPickingListFromHMIWorkArea[j].SupportPianoLegno.YDim;
													WorkAreaState[j].Supporto.ZDim 					:= RequestPickingListFromHMIWorkArea[j].SupportPianoLegno.ZDim;
													WorkAreaOffset[j].Y 							:= OFFSET_POSTAZIONE_LEGNO + RequestPickingListFromHMIWorkArea[j].SupportPianoLegno.YDim/2;//ATTENZIONE!!! per poter lavorare in centro con i supporti pari, questa misura è la distanza tra il riscontro bundle verticale e il centro postazione PARI
												(* Se ho una cassa pianale in ferro su supporto *)
												TELAIO_PIANO:
													WorkAreaState[j].Supporto.Code 					:= ActualPickingListFromHMI[IdxLista].SupportPianoFerro.Code;
													WorkAreaState[j].Supporto.DimBaseUtile		 	:= RequestPickingListFromHMIWorkArea[j].SupportPianoFerro.DimBaseUtile;
													WorkAreaState[j].Supporto.AltezzaDenteRitenuta 	:= RequestPickingListFromHMIWorkArea[j].SupportPianoFerro.ZDim+20;
													WorkAreaState[j].Supporto.DimVertice 			:= RequestPickingListFromHMIWorkArea[j].SupportPianoFerro.DimVertice;
													WorkAreaState[j].Supporto.HMAX 					:= RequestPickingListFromHMIWorkArea[j].SupportPianoFerro.HMAX;
													WorkAreaState[j].Supporto.Tipologia 			:=  e_Tipo_Pallet.CASSA_STANDARD;//ActualPickingListFromHMI[1].Support.Tipologia;
													WorkAreaState[j].Supporto.XDim 					:= RequestPickingListFromHMIWorkArea[j].SupportPianoFerro.XDim;
													WorkAreaState[j].Supporto.YDim 					:= RequestPickingListFromHMIWorkArea[j].SupportPianoFerro.YDim;
													WorkAreaState[j].Supporto.ZDim 					:= RequestPickingListFromHMIWorkArea[j].SupportPianoFerro.ZDim;
													WorkAreaOffset[j].Y 							:= OFFSET_POSTAZIONE_TELAIO - RequestPickingListFromHMIWorkArea[j].SupportPianoFerro.YDim/2;//ATTENZIONE!!! per poter lavorare in centro con i supporti pari, questa misura è la distanza tra il riscontro bundle verticale e il centro postazione PARI
												(* Se ho un bundle *)
												BUNDLE_VERT:
													//WorkAreaState[j].P := ElementiDaDepositare;
													WorkAreaState[j].Supporto.Code 					:= ActualPickingListFromHMI[IdxLista].SupportVertBundle.Code;
													WorkAreaState[j].Supporto.DimBaseUtile		 	:= RequestPickingListFromHMIWorkArea[j].SupportVertBundle.DimBaseUtile;
													WorkAreaState[j].Supporto.AltezzaDenteRitenuta 	:= RequestPickingListFromHMIWorkArea[j].SupportVertBundle.ZDim+20;
													WorkAreaState[j].Supporto.DimVertice 			:= RequestPickingListFromHMIWorkArea[j].SupportVertBundle.DimVertice;
													WorkAreaState[j].Supporto.HMAX 					:= RequestPickingListFromHMIWorkArea[j].SupportVertBundle.HMAX;
													WorkAreaState[j].Supporto.Tipologia 			:= e_Tipo_Pallet.BUNDLE;//ActualPickingListFromHMI.SupportVert.Tipologia;
													WorkAreaState[j].Supporto.XDim 					:= RequestPickingListFromHMIWorkArea[j].SupportVertBundle.XDim;
													WorkAreaState[j].Supporto.YDim 					:= RequestPickingListFromHMIWorkArea[j].SupportVertBundle.YDim;
													WorkAreaState[j].Supporto.ZDim 					:= RequestPickingListFromHMIWorkArea[j].SupportVertBundle.ZDim;
													WorkAreaState[j].Supporto.ZDim_Ext1        		:= WorkAreaState[j].Supporto.ZDim + 20;	
													WorkAreaState[j].Supporto.TipoPianoAppoggio 	:= 1;                      
													WorkAreaState[j].Supporto.AltezzaDenteRitenuta	:= 20; 
													WorkAreaState[j].Supporto.LatoDeposito 			:= 180; 
													//**Lo Que Habia
													WorkAreaOffset[j].Y 							:= 0;
													//Mod 25/&/2025	  
													//WorkAreaOffset[j].Y 		:= ActualPickingListFromHMI[IdxLista].SupportVertBundle.YDim-ActualPickingListFromHMI[IdxLista].SupportVertBundle.DimBaseUtile -40;					
												(* Se ho un A_Frame *)	  
												A_FRAME_VERT:  						
													//WorkAreaState[j].P := ElementiDaDepositare;
													WorkAreaState[j].Supporto.Code 					:= ActualPickingListFromHMI[IdxLista].SupportVertCav.Code;
													WorkAreaState[j].Supporto.DimBaseUtile		 	:= RequestPickingListFromHMIWorkArea[j].SupportVertCav.DimBaseUtile;
													WorkAreaState[j].Supporto.AltezzaDenteRitenuta 	:= RequestPickingListFromHMIWorkArea[j].SupportVertCav.ZDim+20;
													WorkAreaState[j].Supporto.DimVertice 			:= RequestPickingListFromHMIWorkArea[j].SupportVertCav.DimVertice;
													WorkAreaState[j].Supporto.HMAX 					:= RequestPickingListFromHMIWorkArea[j].SupportVertCav.HMAX;
													WorkAreaState[j].Supporto.Tipologia 			:= CAVALLETTO;//ActualPickingListFromHMI.SupportVertCav.Tipologia;
													WorkAreaState[j].Supporto.XDim 					:= RequestPickingListFromHMIWorkArea[j].SupportVertCav.XDim;
													WorkAreaState[j].Supporto.YDim 					:= RequestPickingListFromHMIWorkArea[j].SupportVertCav.YDim;
													WorkAreaState[j].Supporto.ZDim 					:= RequestPickingListFromHMIWorkArea[j].SupportVertCav.ZDim;
													WorkAreaState[j].Supporto.ZDim_Ext1        		:= WorkAreaState[j].Supporto.ZDim + 20;	
													WorkAreaState[j].Supporto.TipoPianoAppoggio 	:= 1;                      
													WorkAreaState[j].Supporto.AltezzaDenteRitenuta	:= 15; 		
													WorkAreaOffset[j].Y 							:= OFFSET_POSTAZIONE_LEGNO + RequestPickingListFromHMIWorkArea[j].SupportVertCav.YDim/2;//ATTENZIONE!!! per poter lavorare in centro con i supporti pari, questa misura è la distanza tra il riscontro bundle verticale e il centro postazione PARI
												   	CoordenadaPasillo0_Y 							:= WorkArea[j].Y +  WorkAreaOffset[j].Y  - Dimensioni_Pinza.Spessore - INGOMBRO_RISCONTRO_BUNDLE - WorkAreaState[j].Supporto.YDim /2 ;
													CoordenadaPasillo180_Y 							:= WorkArea[j].Y + WorkAreaState[j].Supporto.YDim /2 + WorkAreaOffset[j].Y  + Dimensioni_Pinza.Spessore + INGOMBRO_RISCONTRO_FRAME  ;	
												
											END_CASE
													  
											WorkAreaProductionList[j].Support := WorkAreaState[j].Supporto;
										END_IF
									END_IF
									TFClearApprendimento(ADR(WorkAreaState[j].Apprendimento));//Azzeramento apprendimento
								END_FOR
								EXIT; 
						END_CASE // case Pricipal1
					END_IF	//-------->	 //-------> Palet destino
				END_FOR//----------For 1 HMI_WorkAreaDataPicking[i].Destinazione 
				
				Picking.Cmd_CalcolaLista[IdxLista] := TRUE;
				HMI_Forming_Attivazione[IdxLista] := TRUE;//attivo nuova formatura
			END_IF //------------------------------ActualPickingListFromHMI[IdxLista].State = e_StatoWorkOrder.DA_ESEGUIRE 
{endregion }
			 
		    	  


	IF Picking.Cmd_CalcolaLista[IdxLista] AND HMI_Forming_Attivazione[IdxLista] THEN
			idxForm:= IdxLista;		  
		FOR CalFor := Iforstart TO Iforend DO
				CrearFormacion := 1 ; 
				IF CalFor = NumPostazioneDeposito THEN // calcula la formacion para la estacion de piking
					CASE CrearFormacion OF
		  				1:  
							//Ack 
							IF HMI_ErrAckCalcolaFormatura THEN
								HMI_Forming_ErroreCalcoli 					:= 0;
								HMI_ErrAckCalcolaFormatura 					:= FALSE;
								FOR i:= 1 TO MAXFORMING DO
									HMI_ConfermaAttivazioneFormatura[i] 	:= FALSE;
									HMI_Forming_FormaturaAttivata[i] 		:= FALSE;
								END_FOR	 
							END_IF
							
							//Azzeramento comandi in caso di errore
							IF HMI_Forming_ErroreCalcoli <> 0 THEN
								FOR i:=1 TO MAXFORMING DO
									HMI_Forming_Attivazione[i] 				:= FALSE;
									HMI_Forming_Disattivazione[i] 			:= FALSE;
								END_FOR
								HMI_Forming_Calcola 						:= FALSE;
							END_IF
							// borra las estructuras Anteas hacer el calculo
							TFCalcoloFormaturaWA[CalFor].PulisciMemoria := TRUE ;
							HMI_Forming_FormaturaAttivata[idxForm] 		:= FALSE;	
							TFCalcoloFormaturaWA[CalFor]() ;
							CrearFormacion := 2 ; 	  
						2:
								  
							
							IF 	 TFCalcoloFormaturaWA[CalFor].PulisciMemoria AND TFCalcoloFormaturaWA[CalFor].PulisciMemoriaDone THEN 
								// borra La Formacion de la estructura		  
								WorkAreaProductionList[CalFor].Forming := FormingEmpty;
									 
								CASE WorkAreaState[NumPostazioneDeposito].Supporto.Tipologia OF //**Mod
									BUNDLE_VERT:
										TFCalcoloFormaturaWA[CalFor].TipoOrdinamento := 4;//Ordinamento di deposito òato 180°
									A_FRAME_VERT:
										TFCalcoloFormaturaWA[CalFor].TipoOrdinamento := 1;//Ordinamento di deposito, prima un lato poi l'altro	
										TFCalcoloFormaturaWA[CalFor].HabiCalTodasCordenadas := TRUE ;
									ELSE
										TFCalcoloFormaturaWA[CalFor].TipoOrdinamento := 2;//Ordinamento di deposito consecutivo	 
								END_CASE
								(*
									//Valorizzo altezza esterna supporto
									//IF HMI_Forming_Supporto.ZDim_Ext1 = 0 THEN
										HMI_Forming_Supporto.ZDim_Ext1 := HMI_Forming_Supporto.ZDim + HMI_Forming_Supporto.AltezzaDenteRitenuta;
									//END_IF
									//Valorizzo HMAX x tipologia pallet
									IF HMI_Forming_Supporto.Tipologia = PALLET_STANDARD THEN
										HMI_Forming_Supporto.HMAX := HMI_Forming_Supporto.ZDim;
									END_IF 
											  *)
								IF (RequestPickingListFromHMI[1].LayerSequence = 0 OR NOT HMI_AbilitaDepositoFalda)
									AND HMI_Forming_NumeroElementiDaDepositare >0 
								THEN
									//Assegno l'ordine tutto a 1 perchè ho solo lastre	
									FOR i:= 1 TO MAXFORMINGSLAB DO
										//IF i <= HMI_Forming_NumeroElementiDaDepositare THEN
										IF i <= HMI_Forming_NumeroElementiDaDepositare + HMI_NumeroPezziPresentiPostazione[NumPostazioneDeposito] THEN
										//IF i <= 20THEN
											TFCalcoloFormaturaWA[CalFor].TipoElementoDep[i]:= TFCalcoloFormaturaWA[CalFor].TipoElementoDep[i]:= WorkAreaProductionList[CalFor].PElementList[1].PElement.Typology ;
										ELSE
											 TFCalcoloFormaturaWA[CalFor].TipoElementoDep[i] := TERMINATORE;//Settiamo il resto come terminatore
										END_IF
									END_FOR
								ELSE
									//FOR i := 1 TO HMI_Forming_NumeroElementiDaDepositare DO//BY (Request_WorkOrder.LayerSequence+1) DO		  
									FOR i := 1 TO HMI_Forming_NumeroElementiDaDepositare DO//BY (Request_WorkOrder.LayerSequence+1) DO
										IF i MOD 2 = 1 THEN// i <= HMI_Forming_NumeroElementiDaDepositare THEN 
											 TFCalcoloFormaturaWA[CalFor].TipoElementoDep[i]:= WorkAreaProductionList[CalFor].PElementList[i].PElement.Typology ;//Settiamo tipo lastre!!
										ELSE
											 TFCalcoloFormaturaWA[CalFor].TipoElementoDep[i] := FALDA;//Settiamo tipoi falda!
										END_IF
										 	TFCalcoloFormaturaWA[CalFor].TipoElementoDep[i+1] := TERMINATORE;//Settiamo il resto come terminatore
									END_FOR
								END_IF		
								
							
								 TFCalcoloFormaturaWA[CalFor].Materiale[e_Tipo_Elemento_Da_Lavorare.LASTRA]		:= HMI_Forming_LastraDaDepositare; 
								 TFCalcoloFormaturaWA[CalFor].Materiale[e_Tipo_Elemento_Da_Lavorare.FALDA]		:= FaldaDaDepositare;
								 TFCalcoloFormaturaWA[CalFor].Materiale[e_Tipo_Elemento_Da_Lavorare.QUADROTTA]	:= HMI_Forming_LastraDaDepositare;
								 TFCalcoloFormaturaWA[CalFor].Supporto											:= WorkAreaProductionList[CalFor].Support;	//Assegno la tipologia di supporto	  
								
								TFCalcoloFormaturaWA[CalFor].CalcolaFormatura := TRUE; 		//Lancio esecuzione dei calcoli
								MEMSET(ADR(WorkAreaProductionList[CalFor].Forming),0,SIZEOF(WorkAreaProductionList[CalFor].Forming));	//Pulisco la memoria di destinazione
								HMI_Forming_Attivazione[CalFor] := FALSE;
								TFCalcoloFormaturaWA[CalFor].PulisciMemoria := FALSE;  
								TFCalcoloFormaturaWA[CalFor]() ;
							END_IF 
							CrearFormacion := 3 ; 
						3:	
							IF TFCalcoloFormaturaDaLista.CalcolaFormaturaDone OR TFCalcoloFormaturaDaLista.Errore > 0 THEN
								
								TFCalcoloFormaturaWA[CalFor].CalcolaFormatura := FALSE;
								Formacion_De_listaOk[idxForm] := TRUE ;
								IF TFCalcoloFormaturaWA[CalFor].Errore = 0 THEN
									IDFormatura 									:= IDFormatura+1;
									GUIDFormatura 									:= STRING_TO_UINT(concat(UINT_TO_STRING(NUMERO_MACCHINA),UINT_TO_STRING(IDFormatura)));
									HMI_Forming_GUID 								:= GUIDFormatura;
							
									WorkAreaProductionList[CalFor].Forming 			:= TFCalcoloFormaturaDaLista.FormingSlab;
									WorkAreaProductionList[CalFor].Forming.Enable 	:= 1;
									WorkAreaProductionList[CalFor].Forming.Code 	:= HMI_Forming_CodiciAbilitatiFormatura[idxForm].Code;
									WorkAreaProductionList[CalFor].Forming.GUID		:= HMI_Forming_GUID;
											  
									Forming[idxForm] 								:= FormingEmpty;	//Pulisco la memoria di destinazione
									Forming[idxForm] 								:= TFCalcoloFormaturaDaLista.FormingSlab;
									Forming[idxForm].Pallet							:= HMI_Forming_Supporto;
									Forming[idxForm].Enable 						:= 1;
									Forming[idxForm].Code 							:= HMI_Forming_CodiciAbilitatiFormatura[idxForm].Code;
									Forming[idxForm].GUID							:= HMI_Forming_GUID;
											  
									HMI_Forming_IndiceFormaturaAttivata := idxForm;
									HMI_Forming_FormaturaAttivata[idxForm] 	:= TRUE;
									HMI_ConfermaAttivazioneFormatura[idxForm] := TRUE;
									//Valorizzo la struttura del WAPL per ogni elemento da elaborare
											FOR jj := 1 TO MAXELEMENTLIST DO
												IF jj < ElementiElaborati[IdxLista] THEN
													WorkAreaProductionList[NumPostazioneDeposito].PElementList[jj].Stato			:= ELEMENTO_DA_ELABORARE;
													IF Picking.HMI_PareggiaturaLastraAbilitata THEN
														WorkAreaProductionList[NumPostazioneDeposito].PElementList[jj].Pareggiatura := PAREGGIATURA_DA_ESEGUIRE;
													ELSE
														WorkAreaProductionList[NumPostazioneDeposito].PElementList[jj].Pareggiatura := PAREGGIATURA_DISABILITATA;
													END_IF
												ELSE
													WorkAreaProductionList[NumPostazioneDeposito].PElementList[jj].Stato			:= ELEMENTO_NOT_DEFINED;
												END_IF
											END_FOR
								ELSE
									HMI_Forming_ErroreCalcoli := TFCalcoloFormaturaDaLista.Errore;
								END_IF
								HMI_Forming_Attivazione[idxForm] := FALSE;
						END_IF				
								  
					END_CASE	
				END_IF 
					 
//ELSE 
	;
	END_FOR
END_IF
(* 
	ELSE // Todas las formaciones  De coger
					IF HMI_WorkAreaDataPicking[CalFor].NumElementiDaLavorare <> 0 THEN 	  
						CASE CrearFormacion OF
							1: 
								 TFCalcoloFormaturaWA[CalFor].PulisciMemoria 	:= TRUE;
								 TFCalcoloFormaturaWA[CalFor]()	 ;
								 CrearFormacion := 2 ; 
								 ;
							2: 
								IF TFCalcoloFormaturaRT[IdxLista].PulisciMemoriaDone THEN		
									FOR i:= 1 TO MAXFORMINGSLAB DO
										IF i <= 40 THEN
										//IF i <= HMI_Forming_NumeroElementiDaDepositare THEN
											TFCalcoloFormaturaRT[IdxLista].TipoElementoDep[i] := LASTRA;//Settiamo tutte lastre!!
										ELSE
											TFCalcoloFormaturaRT[IdxLista].TipoElementoDep[i] := TERMINATORE;//Settiamo il resto come terminatore
										END_IF
									END_FOR
									TFCalcoloFormaturaWA[CalFor].Materiale[e_Tipo_Elemento_Da_Lavorare.LASTRA].XDim				:= RequestPickingListFromHMIWorkArea[CalFor].SlabDimension.XDim; 
									TFCalcoloFormaturaWA[CalFor].Materiale[e_Tipo_Elemento_Da_Lavorare.LASTRA].YDim				:= RequestPickingListFromHMIWorkArea[CalFor].SlabDimension.YDim; 
									TFCalcoloFormaturaWA[CalFor].Materiale[e_Tipo_Elemento_Da_Lavorare.LASTRA].ZDim				:= RequestPickingListFromHMIWorkArea[CalFor].SlabDimension.ZDim; 
									TFCalcoloFormaturaWA[CalFor].Supporto.Code													:= WorkAreaState[CalFor].Supporto.Code ;
									TFCalcoloFormaturaWA[CalFor].Supporto.XDim													:= WorkAreaState[CalFor].Supporto.XDim;
									TFCalcoloFormaturaWA[CalFor].Supporto.YDim													:= WorkAreaState[CalFor].Supporto.YDim*2;
									TFCalcoloFormaturaWA[CalFor].Supporto.ZDim													:= WorkAreaState[CalFor].Supporto.ZDim;
									TFCalcoloFormaturaWA[CalFor].Supporto.DimBaseUtile											:= WorkAreaState[CalFor].Supporto.DimBaseUtile;
									TFCalcoloFormaturaWA[CalFor].Supporto.DimVertice 											:= WorkAreaState[CalFor].Supporto.DimVertice*2;
									TFCalcoloFormaturaWA[CalFor].Supporto.HMAX 													:= WorkAreaState[CalFor].Supporto.HMAX;
									CASE  WorkAreaState[IdxLista].Supporto.Tipologia OF
										LEGNO_PIANO :
											 			;
										TELAIO_PIANO : 
														;
										BUNDLE_VERT:
											
											TFCalcoloFormaturaWA[CalFor].Supporto.TipoPianoAppoggio 							:= 1;
											TFCalcoloFormaturaWA[CalFor].Supporto.AltezzaDenteRitenuta							:= 15;
											TFCalcoloFormaturaWA[CalFor].Supporto.ZDim_Ext1        								:= TFCalcoloFormaturaWA[CalFor].Supporto.ZDim + TFCalcoloFormaturaWA[CalFor].Supporto.AltezzaDenteRitenuta;
											TFCalcoloFormaturaWA[CalFor].Supporto.Tipologia 									:= BUNDLE;
											TFCalcoloFormaturaWA[CalFor].Supporto.LatoDeposito 									:= 180;
											TFCalcoloFormaturaWA[CalFor].TipoOrdinamento										:= 4;	//Ordinamento di deposito, prima un lato poi l'altro
											
										A_FRAME_VERT:		  
											TFCalcoloFormaturaWA[CalFor].HabiCalTodasCordenadas 								:= TRUE ;
											TFCalcoloFormaturaWA[CalFor].Supporto.TipoPianoAppoggio 							:= 1;
											TFCalcoloFormaturaWA[CalFor].Supporto.AltezzaDenteRitenuta							:= 13;
											TFCalcoloFormaturaWA[CalFor].Supporto.ZDim_Ext1        								:= TFCalcoloFormaturaRT[IdxLista].Supporto.ZDim + TFCalcoloFormaturaRT[IdxLista].Supporto.AltezzaDenteRitenuta;
											TFCalcoloFormaturaWA[CalFor].Supporto.Tipologia 									:= CAVALLETTO;
											TFCalcoloFormaturaWA[CalFor].Supporto.LatoDeposito 									:= 0;
											TFCalcoloFormaturaWA[CalFor].TipoOrdinamento										:= 1;	//Ordinamento di deposito, prima un lato poi l'altro
											 
									END_CASE
									TFCalcoloFormaturaWA[CalFor].CalcolaFormatura 				:= TRUE;//Lancio esecuzione dei calcoli
									MEMSET(ADR(FormaturaWA[CalFor]),0,SIZEOF(FormaturaWA[CalFor]));	//Pulisco la memoria di destinazione
									TFCalcoloFormaturaWA[CalFor].PulisciMemoria 				:= FALSE;
									TFCalcoloFormaturaWA[CalFor]() ;
									CrearFormacion 												:= 3 ; 
								
								
								
							END_IF
									 ;
							3:	
								 IF (TFCalcoloFormaturaRT[IdxLista].CalcolaFormaturaDone OR TFCalcoloFormaturaRT[IdxLista].Errore > 0) AND CalcolaFormaturaTrig2 THEN
										
										TFCalcoloFormaturaWA[CalFor].CalcolaFormatura := FALSE;
										TFFormacionCavalleteCalculada := TFCalcoloFormaturaWA[CalFor] ;
										FormaturaWa[CalFor] := TFCalcoloFormaturaWA[CalFor].FormingSlab;
				
										//CalcolaFormingRT[IdxLista] := TRUE ; // modificacion probar
										IF TFCalcoloFormaturaRT[IdxLista].Errore = 0 THEN
											Formacion_FrameCalOk[idxForm] 		:= TRUE ;
										ELSE
											//CalcolaFormingRT[IdxLista] := TRUE; // original	  
											CalcolaFormingRT2[IdxLista] := TRUE;
										//##############################Fin ##############################################		 
										//#########################Calculo cavaleta##########################################
										END_IF
								END_IF
								 
					END_CASE 
	
				END_IF
			
		END_FOR
	END_IF	 
			
	*)	
//------------------------------------------------------------------------------------------	
					 
				

		
	
				  
					   
		
					   
							
		
			
				  
				
					
				
END_IF			
	
END_FOR	 
	 

	HMI_WorkAreaDataPicking_1_8 := ActualPickingListFromHMI[1].State >= 1;//Ordine postazioni 1..8 in lavoro
		 
	HMI_WorkAreaDataPicking_1_4 := (ActualPickingListFromHMI[2].State >= 1);//Ordine postazioni 1..4 in lavoro
	HMI_WorkAreaDataPicking_5_8 := (ActualPickingListFromHMI[3].State >= 1);//Ordine postazioni 5..8 in lavoro


							  
								   
{endregion}
END_ACTION

ACTION _11_CalcolaListaProduzioneold:
IF MachinePalletizer_TF.IN.Mode.Man AND
	(MachinePalletizer_TF.CmdExe.Code = CmdNOP OR MachinePalletizer_TF.CmdExe.Code = CmdMAN) THEN
	IF Cmd_AzzeraLista THEN
		ActualPickingListFromHMI.State := e_StatoWorkOrder.NON_ESEGUITO;
		FOR i:= 1 TO MAXAREAPRESENT DO	
			TFClearWorkAreaArray(ADR(Workarea),ADR(WorkAreaState),k:=i);
			HMI_WorkAreaDataPicking[i].Destinazione := FALSE;
			HMI_WorkAreaDataPicking[i].NumElementiDaLavorare := 0;
			WorkAreaState[i].P 			:= 1;
			WorkAreaProductionList[i] 	:= ListaEmpty;
			WorkAreaOffset[i].Y 		:= 0;
			HMI_NumeroPezziPresentiPostazione[i] := 0;
			NumeroPezziPresentiPostazioneStart[i] := 0;
		END_FOR	
		HMI_NumeroLastreDepOrdineAttuale := 0; 
		//Disattivazione formatura
		Forming[1] := FormingEmpty;	//Pulisco la formatura selezionata e di consegenza la disattivo
		ActualPickingListFromHMI.State := e_StatoWorkOrder.NON_ESEGUITO;
		//Azzero le liste per le postazioni dove non avviene la pallettizzazione
		WorkAreaProductionList[1].Stato := e_Stato_ListaDiProduzione.LISTA_PROD_ASSENTE;
		WorkAreaProductionList[2].Stato := e_Stato_ListaDiProduzione.LISTA_PROD_ASSENTE;
		WorkAreaProductionList[3].Stato := e_Stato_ListaDiProduzione.LISTA_PROD_ASSENTE;
		WorkAreaProductionList[4].Stato := e_Stato_ListaDiProduzione.LISTA_PROD_ASSENTE;
		WorkAreaProductionList[5].Stato := e_Stato_ListaDiProduzione.LISTA_PROD_ASSENTE;
		WorkAreaProductionList[6].Stato := e_Stato_ListaDiProduzione.LISTA_PROD_ASSENTE;
		WorkAreaProductionList[7].Stato := e_Stato_ListaDiProduzione.LISTA_PROD_ASSENTE;
		WorkAreaProductionList[8].Stato := e_Stato_ListaDiProduzione.LISTA_PROD_ASSENTE;
		ActualPickingListFromHMI.SlabNumber 		:= 0;
		ActualPickingListFromHMI.SlabDimension.XDim := 0;
		ActualPickingListFromHMI.SlabDimension.YDim := 0;
		ActualPickingListFromHMI.SlabDimension.ZDim := 0;
		ActualPickingListFromHMI.Support 			:= SupportDataEmpty;
		
		HMI_ErroreCalcoloLista 		:= 0;
		Picking.Cmd_CalcolaLista 	:= FALSE;
		HMI_Forming_Attivazione[1] 	:= FALSE;//attivo nuova formatura
		
		Cmd_AzzeraLista := FALSE;
		//Ack 
		//IF HMI_ErrAckCalcolaFormatura THEN
			HMI_Forming_ErroreCalcoli := 0;
			HMI_ErrAckCalcolaFormatura := FALSE;
			FOR i:= 1 TO MAXFORMING DO
				HMI_Forming_FormaturaAttivata[i] := FALSE;
			END_FOR
		//END_IF
		CalcolaFormaturaTrig := FALSE;
	END_IF
	
	IF Cmd_AttivaLista AND ActualPickingListFromHMI.State <> e_StatoWorkOrder.IN_ESECUZIONE THEN
		ElementiDaDepositare   :=0;
		HMI_ErroreCalcoloLista := 0;
		HMI_NumeroLastreDepOrdineAttuale := 0;
		FOR i:= 1 TO MAXAREAPRESENT DO	
			//HMI_WorkAreaDataPicking[i].Destinazione := FALSE;
			//HMI_WorkAreaDataPicking[i].NumElementiDaLavorare := 0;
			WorkAreaState[i].P := 1;
			WorkAreaProductionList[i] := ListaEmpty;
		END_FOR	 
		
		FOR i:= 1 TO MAXAREAPRESENT DO	
			IF NOT HMI_WorkAreaDataPicking[i].Destinazione THEN
				ElementiDaDepositare := ElementiDaDepositare+HMI_WorkAreaDataPicking[i].NumElementiDaLavorare;
				WorkAreaState[i].P := HMI_WorkAreaDataPicking[i].NumElementiDaLavorare +1;
				IF HMI_WorkAreaDataPicking[i].Vertical THEN
					WorkareaState[i].Supporto.Tipologia := BUNDLE;
				ELSE
					WorkareaState[i].Supporto.Tipologia := CASSA_STANDARD;
				END_IF
			ELSE
				NumPostazioneDeposito := i;
				HMI_WorkAreaDataPicking[NumPostazioneDeposito].NumElementiDaLavorare := RequestPickingListFromHMI.SlabNumber;
				IF HMI_WorkAreaDataPicking[i].Vertical THEN
					WorkareaState[i].Supporto.Tipologia := BUNDLE;
				ELSE
					WorkareaState[i].Supporto.Tipologia := CASSA_STANDARD;
				END_IF
			END_IF
			HMI_NumeroPezziPresentiPostazione[i] := WorkAreaState[i].P -1;
		END_FOR
	
		IF ElementiDaDepositare <= HMI_WorkAreaDataPicking[NumPostazioneDeposito].NumElementiDaLavorare THEN
			ActualPickingListFromHMI 		:= RequestPickingListFromHMI;
			ActualPickingListFromHMI.State 	:= e_StatoWorkOrder.DA_ESEGUIRE;
		ELSE
			HMI_ErroreCalcoloLista := 1;
		END_IF
		Cmd_AttivaLista 				:= FALSE;
	ELSE
		Cmd_AttivaLista 				:= FALSE;
	END_IF
	
	//attivazione lista di picking
	IF ActualPickingListFromHMI.State = e_StatoWorkOrder.DA_ESEGUIRE THEN
		ListaInEsecuzione := FALSE;
		NumeroListaInEsecuzione := 0;
	
		(* Inserimento sequenza di prelievo dalle postazioni in base al quello che l'operatore ha editato da HMI*)
		ElementiDaDepositare := 0;
		ElementiElaborati    := 1;
		NumPostazioneDeposito := 0;
		//FOR i:= 1 TO MAXAREAPRESENT DO
		//	WorkAreaState[i].P := 1;
		//END_FOR		
		
		FOR i:= 1 TO MAXAREAPRESENT DO
			IF HMI_WorkAreaDataPicking[i].Destinazione THEN
				NumPostazioneDeposito := i;
				HMI_WorkAreaDataPicking[NumPostazioneDeposito].NumElementiDaLavorare 	:= RequestPickingListFromHMI.SlabNumber;
				IF NOT HMI_WorkAreaDataPicking[NumPostazioneDeposito].Vertical THEN //Se NON ho deposito verticale
					WorkAreaState[NumPostazioneDeposito].Supporto.Code 						:= ActualPickingListFromHMI.Support.Code;
					WorkAreaState[NumPostazioneDeposito].Supporto.AltezzaDenteRitenuta 		:= ActualPickingListFromHMI.Support.DimBaseUtile;
					WorkAreaState[NumPostazioneDeposito].Supporto.DimVertice 				:= ActualPickingListFromHMI.Support.DimVertice;
					WorkAreaState[NumPostazioneDeposito].Supporto.HMAX 						:= ActualPickingListFromHMI.Support.HMAX;
					WorkAreaState[NumPostazioneDeposito].Supporto.Tipologia 				:= CASSA_STANDARD;//ActualPickingListFromHMI.Support.Tipologia;
					WorkAreaState[NumPostazioneDeposito].Supporto.XDim 						:= ActualPickingListFromHMI.Support.XDim;
					WorkAreaState[NumPostazioneDeposito].Supporto.YDim 						:= ActualPickingListFromHMI.Support.YDim;
					WorkAreaState[NumPostazioneDeposito].Supporto.ZDim 						:= ActualPickingListFromHMI.Support.ZDim;
					WorkAreaOffset[NumPostazioneDeposito].Y 								:= 1315;//ATTENZIONE!!! per poter lavorare in centro con i supporti pari, questa misura è la distanza tra il riscontro bundle verticale e il centro postazione PARI
					
					FOR j := 1 TO MAXAREAPRESENT DO
						IF NOT HMI_WorkAreaDataPicking[j].Destinazione THEN
							IF HMI_WorkAreaDataPicking[j].NumElementiDaLavorare >= 1 THEN
								ElementiDaDepositare := ElementiElaborati + HMI_WorkAreaDataPicking[j].NumElementiDaLavorare;
								FOR k := ElementiElaborati TO ElementiDaDepositare-1 DO	
									WorkAreaProductionList[NumPostazioneDeposito].PElementList[k].WA_PRELIEVO := j;
									WorkAreaProductionList[NumPostazioneDeposito].PElementList[k].WA_DEPOSITO := i;	
									ElementiElaborati := ElementiElaborati+1; 
								END_FOR
								IF NOT HMI_WorkAreaDataPicking[j].Vertical THEN
									WorkAreaState[j].Supporto.Code 					:= ActualPickingListFromHMI.Support.Code;
									WorkAreaState[j].Supporto.DimBaseUtile		 	:= ActualPickingListFromHMI.Support.DimBaseUtile;
									WorkAreaState[j].Supporto.AltezzaDenteRitenuta 	:= ActualPickingListFromHMI.Support.ZDim+20;
									WorkAreaState[j].Supporto.DimVertice 			:= ActualPickingListFromHMI.Support.DimVertice;
									WorkAreaState[j].Supporto.HMAX 					:= ActualPickingListFromHMI.Support.HMAX;
									WorkAreaState[j].Supporto.Tipologia 			:= ActualPickingListFromHMI.Support.Tipologia;
									WorkAreaState[j].Supporto.XDim 					:= ActualPickingListFromHMI.Support.XDim;
									WorkAreaState[j].Supporto.YDim 					:= ActualPickingListFromHMI.Support.YDim;
									WorkAreaState[j].Supporto.ZDim 					:= ActualPickingListFromHMI.Support.ZDim;
									WorkAreaOffset[j].Y 							:= 1315;//ATTENZIONE!!! per poter lavorare in centro con i supporti pari, questa misura è la distanza tra il riscontro bundle verticale e il centro postazione PARI
								ELSE
									//WorkAreaState[j].P := ElementiDaDepositare;
									WorkAreaState[j].Supporto.Code 					:= ActualPickingListFromHMI.SupportVert.Code;
									WorkAreaState[j].Supporto.DimBaseUtile		 	:= ActualPickingListFromHMI.SupportVert.DimBaseUtile;
									WorkAreaState[j].Supporto.AltezzaDenteRitenuta 	:= ActualPickingListFromHMI.Support.ZDim+20;
									WorkAreaState[j].Supporto.DimVertice 			:= ActualPickingListFromHMI.SupportVert.DimVertice;
									WorkAreaState[j].Supporto.HMAX 					:= ActualPickingListFromHMI.SupportVert.HMAX;
									WorkAreaState[j].Supporto.Tipologia 			:= 5;//ActualPickingListFromHMI.SupportVert.Tipologia;
									WorkAreaState[j].Supporto.XDim 					:= ActualPickingListFromHMI.SupportVert.XDim;
									WorkAreaState[j].Supporto.YDim 					:= ActualPickingListFromHMI.SupportVert.YDim;
									WorkAreaState[j].Supporto.ZDim 					:= ActualPickingListFromHMI.SupportVert.ZDim;
									WorkAreaState[j].Supporto.ZDim_Ext1        		:= WorkAreaState[j].Supporto.ZDim + 20;					
								END_IF
							END_IF
						END_IF
						TFClearApprendimento(ADR(WorkAreaState[j].Apprendimento));//Azzeramento apprendimento
					END_FOR
					EXIT; 
				ELSE //Se ho deposito verticale
					WorkAreaState[NumPostazioneDeposito].Supporto.Code 						:= ActualPickingListFromHMI.SupportVert.Code;
					WorkAreaState[NumPostazioneDeposito].Supporto.DimBaseUtile		 		:= ActualPickingListFromHMI.SupportVert.DimBaseUtile;
					WorkAreaState[NumPostazioneDeposito].Supporto.DimVertice 				:= ActualPickingListFromHMI.SupportVert.DimVertice;
					WorkAreaState[NumPostazioneDeposito].Supporto.HMAX 						:= ActualPickingListFromHMI.SupportVert.HMAX;
					WorkAreaState[NumPostazioneDeposito].Supporto.Tipologia 				:= BUNDLE;//ActualPickingListFromHMI.SupportVert.Tipologia;
					WorkAreaState[NumPostazioneDeposito].Supporto.XDim 						:= ActualPickingListFromHMI.SupportVert.XDim;
					WorkAreaState[NumPostazioneDeposito].Supporto.YDim 						:= ActualPickingListFromHMI.SupportVert.YDim;
					WorkAreaState[NumPostazioneDeposito].Supporto.ZDim 						:= ActualPickingListFromHMI.SupportVert.ZDim;
					FOR j := 1 TO MAXAREAPRESENT DO
						IF NOT HMI_WorkAreaDataPicking[j].Destinazione THEN
							IF HMI_WorkAreaDataPicking[j].NumElementiDaLavorare >= 1 THEN
								ElementiDaDepositare := ElementiElaborati + HMI_WorkAreaDataPicking[j].NumElementiDaLavorare;
								FOR k := ElementiElaborati TO ElementiDaDepositare-1 DO	
									WorkAreaProductionList[NumPostazioneDeposito].PElementList[k].WA_PRELIEVO := j;
									WorkAreaProductionList[NumPostazioneDeposito].PElementList[k].WA_DEPOSITO := i;	
									ElementiElaborati := ElementiElaborati+1; 
								END_FOR
								IF NOT HMI_WorkAreaDataPicking[j].Vertical THEN
									WorkAreaState[j].Supporto.Code 					:= ActualPickingListFromHMI.Support.Code;
									WorkAreaState[j].Supporto.DimBaseUtile		 	:= ActualPickingListFromHMI.Support.DimBaseUtile;
									WorkAreaState[j].Supporto.AltezzaDenteRitenuta 		:= ActualPickingListFromHMI.Support.ZDim+20;
									WorkAreaState[j].Supporto.DimVertice 			:= ActualPickingListFromHMI.Support.DimVertice;
									WorkAreaState[j].Supporto.HMAX 					:= ActualPickingListFromHMI.Support.HMAX;
									WorkAreaState[j].Supporto.Tipologia 			:= ActualPickingListFromHMI.Support.Tipologia;
									WorkAreaState[j].Supporto.XDim 					:= ActualPickingListFromHMI.Support.XDim;
									WorkAreaState[j].Supporto.YDim 					:= ActualPickingListFromHMI.Support.YDim;
									WorkAreaState[j].Supporto.ZDim 					:= ActualPickingListFromHMI.Support.ZDim;
									WorkAreaOffset[j].Y 							:= 1315;//ATTENZIONE!!! per poter lavorare in centro con i supporti pari, questa misura è la distanza tra il riscontro bundle verticale e il centro postazione PARI
								ELSE
									//WorkAreaState[j].P := ElementiDaDepositare;
									WorkAreaState[j].Supporto.Code 					:= ActualPickingListFromHMI.SupportVert.Code;
									WorkAreaState[j].Supporto.DimBaseUtile 			:= ActualPickingListFromHMI.SupportVert.DimBaseUtile;
									WorkAreaState[j].Supporto.AltezzaDenteRitenuta 	:= ActualPickingListFromHMI.Support.ZDim+20;
									WorkAreaState[j].Supporto.DimVertice 			:= ActualPickingListFromHMI.SupportVert.DimVertice;
									WorkAreaState[j].Supporto.HMAX 					:= ActualPickingListFromHMI.SupportVert.HMAX;
									WorkAreaState[j].Supporto.Tipologia 			:= 5;//ActualPickingListFromHMI.SupportVert.Tipologia;
									WorkAreaState[j].Supporto.XDim 					:= ActualPickingListFromHMI.SupportVert.XDim;
									WorkAreaState[j].Supporto.YDim 					:= ActualPickingListFromHMI.SupportVert.YDim;
									WorkAreaState[j].Supporto.ZDim 					:= ActualPickingListFromHMI.SupportVert.ZDim;
									WorkAreaState[j].Supporto.ZDim_Ext1        		:= WorkAreaState[j].Supporto.ZDim + 20;
								END_IF
							END_IF
						END_IF
						TFClearApprendimento(ADR(WorkAreaState[j].Apprendimento));//Azzeramento apprendimento
					END_FOR
					EXIT; 
				END_IF
			END_IF
		END_FOR
		
		Picking.Cmd_CalcolaLista := TRUE;
		HMI_Forming_Attivazione[1] := TRUE;//attivo nuova formatura
	END_IF
	
	//una volta calcolata la lista per stabilire le postazioni di prelievo e quella di deposito, calcolo la formatura della postazione di deposito
	IF Picking.Cmd_CalcolaLista THEN
		IF NOT HMI_WorkAreaDataPicking[NumPostazioneDeposito].Vertical THEN
			HMI_Formatura.HMI_Forming_Supporto.Code				:= RequestPickingListFromHMI.Support.Code;
			HMI_Formatura.HMI_Forming_Supporto.XDim				:= RequestPickingListFromHMI.Support.XDim;
			HMI_Formatura.HMI_Forming_Supporto.YDim				:= RequestPickingListFromHMI.Support.YDim;
			HMI_Formatura.HMI_Forming_Supporto.ZDim				:= RequestPickingListFromHMI.Support.ZDim;
			HMI_Formatura.HMI_Forming_Supporto.DimBaseUtile		:= RequestPickingListFromHMI.Support.DimBaseUtile;
			HMI_Formatura.HMI_Forming_Supporto.DimVertice 		:= RequestPickingListFromHMI.Support.DimVertice;
			HMI_Formatura.HMI_Forming_Supporto.HMAX 			:= RequestPickingListFromHMI.Support.HMAX;
			HMI_Formatura.HMI_Forming_Supporto.Tipologia		:= RequestPickingListFromHMI.Support.Tipologia;
		ELSE
			HMI_Formatura.HMI_Forming_Supporto.Code				:= RequestPickingListFromHMI.SupportVert.Code;
			HMI_Formatura.HMI_Forming_Supporto.XDim				:= RequestPickingListFromHMI.Supportvert.XDim;
			HMI_Formatura.HMI_Forming_Supporto.YDim				:= RequestPickingListFromHMI.Supportvert.YDim*2;
			HMI_Formatura.HMI_Forming_Supporto.ZDim				:= RequestPickingListFromHMI.Supportvert.ZDim;
			HMI_Formatura.HMI_Forming_Supporto.TipoPianoAppoggio := 1;
			HMI_Formatura.HMI_Forming_Supporto.AltezzaDenteRitenuta		:= 20;
			HMI_Formatura.HMI_Forming_Supporto.ZDim_Ext1        := HMI_Formatura.HMI_Forming_Supporto.ZDim +	HMI_Formatura.HMI_Forming_Supporto.AltezzaDenteRitenuta;
			HMI_Formatura.HMI_Forming_Supporto.DimBaseUtile		:= RequestPickingListFromHMI.Supportvert.DimBaseUtile;
			HMI_Formatura.HMI_Forming_Supporto.DimVertice 		:= RequestPickingListFromHMI.Supportvert.DimVertice*2;
			HMI_Formatura.HMI_Forming_Supporto.HMAX 			:= RequestPickingListFromHMI.Supportvert.HMAX;
			HMI_Formatura.HMI_Forming_Supporto.Tipologia 		:= BUNDLE;
			HMI_Formatura.HMI_Forming_Supporto.LatoDeposito 	:= 180;
		END_IF
		//
		HMI_Formatura.HMI_Forming_LastraDaDepositare.XDim		:= RequestPickingListFromHMI.SlabDimension.XDim;
		HMI_Formatura.HMI_Forming_LastraDaDepositare.YDim		:= RequestPickingListFromHMI.SlabDimension.YDim;
		HMI_Formatura.HMI_Forming_LastraDaDepositare.ZDim		:= RequestPickingListFromHMI.SlabDimension.ZDim;
		
		HMI_Formatura.HMI_Forming_CodiciAbilitatiFormatura[1].Code[1] := 1;
		
		FaldaDaDepositare.TypologyCode := RequestPickingListFromHMI.Layer.Tipologia;
		
		FaldaDaDepositare.XDim := RequestPickingListFromHMI.Layer.XDim;
		FaldaDaDepositare.YDim := RequestPickingListFromHMI.Layer.YDim;
		FaldaDaDepositare.ZDim := RequestPickingListFromHMI.Layer.ZDim;
		
		//Vado ad assegnare il numero giusto di elementi a seconda se è presente o meno la falda 
		IF (RequestPickingListFromHMI.LayerSequence = 1 AND HMI_AbilitaDepositoFalda) AND RequestPickingListFromHMI.Support.Tipologia <> CAVALLETTO AND RequestPickingListFromHMI.Support.Tipologia <> BUNDLE THEN 
			HMI_Formatura.HMI_Forming_NumeroElementiDaDepositare	:= TO_UINT(2*RequestPickingListFromHMI.SlabNumber - 1);
		ELSE 
			HMI_Formatura.HMI_Forming_NumeroElementiDaDepositare	:= TO_UINT(RequestPickingListFromHMI.SlabNumber);
		END_IF
		
		//Ack 
		IF HMI_ErrAckCalcolaFormatura THEN
			HMI_Forming_ErroreCalcoli := 0;
			HMI_ErrAckCalcolaFormatura := FALSE;
			FOR i:= 1 TO MAXFORMING DO
				HMI_Forming_FormaturaAttivata[i] := FALSE;
			END_FOR
		END_IF
		
		//Azzeramento comandi in caso di errore
		IF HMI_Forming_ErroreCalcoli <> 0 THEN
			FOR i:=1 TO MAXFORMING DO
				HMI_Forming_Attivazione[i] 		:= FALSE;
				HMI_Forming_Disattivazione[i] 	:= FALSE;
			END_FOR
			HMI_Forming_Calcola 			:= FALSE;
		END_IF
		
		//Valorizzo altezza esterna supporto
		//IF HMI_Forming_Supporto.ZDim_Ext1 = 0 THEN
			HMI_Forming_Supporto.ZDim_Ext1 := HMI_Forming_Supporto.ZDim + HMI_Forming_Supporto.AltezzaDenteRitenuta;
		//END_IF
		//Valorizzo HMAX x tipologia pallet
		IF HMI_Forming_Supporto.Tipologia = PALLET_STANDARD THEN
			HMI_Forming_Supporto.HMAX := HMI_Forming_Supporto.ZDim;
		END_IF
		
		//Attivazione
		//FOR i:= 1 TO MAXFORMING DO
			idxForm:=1;//forzo a 1 la formatura da attivare
			IF HMI_Forming_Attivazione[idxForm] AND idxForm <=2 THEN
				Forming[idxForm] := FormingEmpty;
				IF NOT CalcolaFormaturaTrig  THEN
					HMI_Forming_FormaturaAttivata[idxForm] 	:= FALSE;
					TFCalcoloFormaturaDaLista.PulisciMemoria 	:= TRUE;
					IF TFCalcoloFormaturaDaLista.PulisciMemoriaDone THEN	
						HMI_Forming_ErroreCalcoli := 0;
						
						IF RequestPickingListFromHMI.LayerSequence = 0 OR NOT HMI_AbilitaDepositoFalda THEN
							//Assegno l'ordine tutto a 1 perchè ho solo lastre	
							FOR i:= 1 TO MAXFORMINGSLAB DO
								IF i <= HMI_Forming_NumeroElementiDaDepositare THEN
									TFCalcoloFormaturaDaLista.TipoElementoDep[i] := LASTRA;//Settiamo tutte lastre!!
								ELSE
									TFCalcoloFormaturaDaLista.TipoElementoDep[i] := TERMINATORE;//Settiamo il resto come terminatore
								END_IF
							END_FOR
						ELSE
							FOR i := 1 TO HMI_Forming_NumeroElementiDaDepositare DO//BY (Request_WorkOrder.LayerSequence+1) DO
								IF i MOD 2 = 1 THEN// i <= HMI_Forming_NumeroElementiDaDepositare THEN 
									TFCalcoloFormaturaDaLista.TipoElementoDep[i] := LASTRA;//Settiamo tipo lastre!!
								ELSE
									TFCalcoloFormaturaDaLista.TipoElementoDep[i] := FALDA;//Settiamo tipoi falda!
								END_IF
								TFCalcoloFormaturaDaLista.TipoElementoDep[i+1] := TERMINATORE;//Settiamo il resto come terminatore
							END_FOR
						END_IF	
						FOR i := HMI_Forming_NumeroElementiDaDepositare+1 TO MAXFORMINGSLAB DO
							TFCalcoloFormaturaDaLista.TipoElementoDep[i] := TERMINATORE;//Settiamo il resto come terminatore
						END_FOR
							
						TFCalcoloFormaturaDaLista.Materiale[e_Tipo_Elemento_Da_Lavorare.LASTRA]		:= HMI_Forming_LastraDaDepositare; 
						TFCalcoloFormaturaDaLista.Materiale[e_Tipo_Elemento_Da_Lavorare.FALDA]		:= FaldaDaDepositare;
						TFCalcoloFormaturaDaLista.Materiale[e_Tipo_Elemento_Da_Lavorare.QUADROTTA]	:= HMI_Forming_LastraDaDepositare;
						TFCalcoloFormaturaDaLista.Supporto											:= HMI_Forming_Supporto;	//Assegno la tipologia di supporto
						IF HMI_WorkAreaDataPicking[NumPostazioneDeposito].Vertical THEN//Se sono in deposito verticale -> sono sul bundle...
							TFCalcoloFormaturaDaLista.TipoOrdinamento									:= 4;//Ordinamento di deposito, prima un lato poi l'altro
						ELSE
							TFCalcoloFormaturaDaLista.TipoOrdinamento									:= 2;//Ordinamento di deposito, prima un lato poi l'altro
						END_IF
						TFCalcoloFormaturaDaLista.CalcolaFormatura := TRUE; 		//Lancio esecuzione dei calcoli
						MEMSET(ADR(HMI_Forming_FormaturaCalcolata),0,SIZEOF(HMI_Forming_FormaturaCalcolata));	//Pulisco la memoria di destinazione
						CalcolaFormaturaTrig := TRUE;
						HMI_Forming_Attivazione[i] := FALSE;
						TFCalcoloFormaturaDaLista.PulisciMemoria := FALSE;
					END_IF
				ELSIF (TFCalcoloFormaturaDaLista.CalcolaFormaturaDone OR TFCalcoloFormaturaDaLista.Errore > 0) AND CalcolaFormaturaTrig THEN
					TFCalcoloFormaturaDaLista.CalcolaFormatura := FALSE;
					IF TFCalcoloFormaturaDaLista.Errore = 0 THEN
						IDFormatura 			:= IDFormatura+1;
						GUIDFormatura 			:= STRING_TO_UINT(concat(UINT_TO_STRING(NUMERO_MACCHINA),UINT_TO_STRING(IDFormatura)));
						HMI_Forming_GUID 		:= GUIDFormatura;
				
						HMI_Forming_FormaturaCalcolata 		:= TFCalcoloFormaturaDaLista.FormingSlab;
						Forming[idxForm] 							:= FormingEmpty;	//Pulisco la memoria di destinazione
						Forming[idxForm] 							:= TFCalcoloFormaturaDaLista.FormingSlab;
						Forming[idxForm].Enable 					:= 1;
						Forming[idxForm].Code 					:= HMI_Forming_CodiciAbilitatiFormatura[idxForm].Code;
						Forming[idxForm].GUID						:= HMI_Forming_GUID;
						Forming[idxForm].Pallet					:= HMI_Forming_Supporto;
						HMI_Forming_IndiceFormaturaAttivata := idxForm;
						HMI_Forming_FormaturaAttivata[idxForm] 	:= TRUE;
						//Valorizzo la struttura del WAPL per ogni elemento da elaborare
						FOR j := 1 TO MAXELEMENTLIST DO
							IF j < ElementiElaborati THEN
								WorkAreaProductionList[NumPostazioneDeposito].PElementList[j].PElement 		:= TFCalcoloFormaturaDaLista.FormingSlab.PElement[j];	
								WorkAreaProductionList[NumPostazioneDeposito].PElementList[j].Stato			:= ELEMENTO_DA_ELABORARE;
							
								IF Picking.HMI_PareggiaturaLastraAbilitata THEN
									WorkAreaProductionList[NumPostazioneDeposito].PElementList[j].Pareggiatura := PAREGGIATURA_DA_ESEGUIRE;
								ELSE
									WorkAreaProductionList[NumPostazioneDeposito].PElementList[j].Pareggiatura := PAREGGIATURA_DISABILITATA;
								END_IF
							ELSE
								WorkAreaProductionList[NumPostazioneDeposito].PElementList[j].Stato			:= ELEMENTO_NOT_DEFINED;
							END_IF
						END_FOR
					ELSE
						HMI_Forming_ErroreCalcoli := TFCalcoloFormaturaDaLista.Errore;
					END_IF
					CalcolaFormaturaTrig := FALSE;
					HMI_Forming_Attivazione[idxForm] := FALSE;
				END_IF
			ELSIF HMI_Forming_Attivazione[idxForm] THEN
				memset(destAddr:=ADR(TFCalcoloFormaturaDaLista.Errore),fillByte:=(UINT_TO_USINT(ErrNumeroMassimoFormatureAmmesse)),n:=SIZEOF(TFCalcoloFormaturaDaLista.Errore));
			END_IF
		
			//Disattivazione formatura
			IF HMI_Forming_Disattivazione[idxForm] THEN
				HMI_Forming_Disattivazione[idxForm] := FALSE;
				Forming[idxForm] := FormingEmpty;	//Pulisco la formatura selezionata e di consegenza la disattivo
			END_IF
				
		//END_FOR
		
		(* Metto in stato di esecuzione il nuovo W.O. se tutto si è attivato *)
		IF HMI_Forming_FormaturaAttivata[1] THEN
			ActualPickingListFromHMI.State := e_StatoWorkOrder.IN_ESECUZIONE;
			//Azzero le liste per le postazioni dove non avviene la pallettizzazione
			WorkAreaProductionList[1].Stato := e_Stato_ListaDiProduzione.LISTA_PROD_ASSENTE;
			WorkAreaProductionList[2].Stato := e_Stato_ListaDiProduzione.LISTA_PROD_ASSENTE;
			WorkAreaProductionList[3].Stato := e_Stato_ListaDiProduzione.LISTA_PROD_ASSENTE;
			WorkAreaProductionList[4].Stato := e_Stato_ListaDiProduzione.LISTA_PROD_ASSENTE;
			WorkAreaProductionList[5].Stato := e_Stato_ListaDiProduzione.LISTA_PROD_ASSENTE;
			WorkAreaProductionList[6].Stato := e_Stato_ListaDiProduzione.LISTA_PROD_ASSENTE;
			WorkAreaProductionList[7].Stato := e_Stato_ListaDiProduzione.LISTA_PROD_ASSENTE;
			WorkAreaProductionList[8].Stato := e_Stato_ListaDiProduzione.LISTA_PROD_ASSENTE;
			WorkAreaProductionList[NumPostazioneDeposito].Support := Forming[idxForm].Pallet;
			WorkAreaProductionList[NumPostazioneDeposito].Stato := LISTA_PROD_DA_ESEGUIRE;
			Picking.Cmd_CalcolaLista := FALSE;
			HMI_Forming_FormaturaAttivata[1] := FALSE;
			CalcolaFormingRT := TRUE;
		END_IF
	END_IF	
	TFCalcoloFormaturaDaLista();
END_IF	

//verifico che la lista sia in esecuzione o terminata
IF NOT ListaInEsecuzione THEN
	FOR i := 1 TO MAXAREAPRESENT DO	
		IF WorkAreaProductionList[i].Stato = e_Stato_ListaDiProduzione.LISTA_PROD_IN_ESECUZIONE THEN
			ListaInEsecuzione := TRUE;
			EXIT;	
		END_IF
	END_FOR
ELSE
	FOR i := 1 TO MAXAREAPRESENT DO	
		IF WorkAreaProductionList[i].Stato = e_Stato_ListaDiProduzione.LISTA_PROD_ESEGUITA THEN
			ListaInEsecuzione := FALSE;
			EXIT;	
		END_IF
	END_FOR
END_IF

//



FOR i := 1 TO MAXAREAPRESENT DO	
		
	IF NumeroPezziPresentiPostazioneStart[i] = 0 AND WorkAreaState[i].P > 1 THEN
		NumeroPezziPresentiPostazioneStart[i] := TO_UINT(WorkAreaState[i].P);
	END_IF

	IF NOT HMI_WorkAreaDataPicking[i].Destinazione THEN
		IF HMI_WorkAreaDataPicking[i].NumElementiDaLavorare > 0 THEN
			//IF HMI_WorkAreaDataPicking[i].NumElementiDaLavorare >= TO_UINT(WorkAreaState[i].P)-1 THEN
			//	HMI_NumeroLastreRimanentiOrdineAttuale[i] := HMI_WorkAreaDataPicking[i].NumElementiDaLavorare - TO_UINT(WorkAreaState[i].P);
			//ELSE
			//	HMI_NumeroLastreRimanentiOrdineAttuale[i] := 0;
			//END_IF
			IF HMI_WorkAreaDataPicking[i].NumElementiDaLavorare - (TO_UINT(WorkAreaState[i].P) - NumeroPezziPresentiPostazioneStart[i]) > 0 THEN
				HMI_NumeroLastreRimanentiOrdineAttuale[i] := MIN(HMI_WorkAreaDataPicking[i].NumElementiDaLavorare,HMI_WorkAreaDataPicking[i].NumElementiDaLavorare - 
															(NumeroPezziPresentiPostazioneStart[i] - TO_UINT(WorkAreaState[i].P)));
			ELSE
				HMI_NumeroLastreRimanentiOrdineAttuale[i] := 0;
			END_IF
		ELSE
			HMI_NumeroLastreRimanentiOrdineAttuale[i] := 0;
		END_IF
	ELSE
		IF NumeroPezziPresentiPostazioneStart[i] < (TO_UINT(WorkAreaState[i].P)) AND NumeroPezziPresentiPostazioneStart[i]>0 THEN
			HMI_NumeroLastreRimanentiOrdineAttuale[i] := TO_UINT(WorkAreaState[i].P) - NumeroPezziPresentiPostazioneStart[i]+1;
		ELSE
			HMI_NumeroLastreRimanentiOrdineAttuale[i] := 0;
		END_IF
	END_IF
	IF (WorkAreaProductionList[i].Stato = e_Stato_ListaDiProduzione.LISTA_PROD_IN_ESECUZIONE OR WorkAreaProductionList[i].Stato = e_Stato_ListaDiProduzione.LISTA_PROD_ESEGUITA) AND WorkAreaState[i].P > 1 THEN
		HMI_NumeroLastreDepOrdineAttuale := TO_UINT(WorkAreaState[i].P-1);
		IF NumeroPezziPresentiPostazioneStart[i] < (TO_UINT(WorkAreaState[i].P)) AND NumeroPezziPresentiPostazioneStart[i]>0 THEN
			HMI_NumeroLastreDepOrdineAttuale := TO_UINT(WorkAreaState[i].P) - NumeroPezziPresentiPostazioneStart[i];
		ELSE
			HMI_NumeroLastreDepOrdineAttuale := 0;
		END_IF
	END_IF	
END_FOR

//trasferisco i valori alla variabile in lettura x HMI
MEMCPY(destAddr:=ADR(HMI_WorkAreaProductionList),srcAddr:=ADR(WorkAreaProductionList),n:=SIZEOF(HMI_WorkAreaProductionList));
	
IF CalcolaFormingRT THEN
	IF NOT CalcolaFormaturaTrig2 THEN
	///////////////////////////
		TFCalcoloFormaturaRT.PulisciMemoria 	:= TRUE;
		IF TFCalcoloFormaturaRT.PulisciMemoriaDone THEN		
			FOR i:= 1 TO MAXFORMINGSLAB DO
				IF i <= 50 THEN
					TFCalcoloFormaturaRT.TipoElementoDep[i] := LASTRA;//Settiamo tutte lastre!!
				ELSE
					TFCalcoloFormaturaRT.TipoElementoDep[i] := TERMINATORE;//Settiamo il resto come terminatore
				END_IF
			END_FOR
			TFCalcoloFormaturaRT.Materiale[e_Tipo_Elemento_Da_Lavorare.LASTRA].XDim		:= RequestPickingListFromHMI.SlabDimension.XDim; 
			TFCalcoloFormaturaRT.Materiale[e_Tipo_Elemento_Da_Lavorare.LASTRA].YDim		:= RequestPickingListFromHMI.SlabDimension.YDim; 
			TFCalcoloFormaturaRT.Materiale[e_Tipo_Elemento_Da_Lavorare.LASTRA].ZDim		:= RequestPickingListFromHMI.SlabDimension.ZDim; 
			TFCalcoloFormaturaRT.Supporto.Code					:= RequestPickingListFromHMI.SupportVert.Code;
			TFCalcoloFormaturaRT.Supporto.XDim					:= RequestPickingListFromHMI.Supportvert.XDim;
			TFCalcoloFormaturaRT.Supporto.YDim					:= RequestPickingListFromHMI.Supportvert.YDim*2;
			TFCalcoloFormaturaRT.Supporto.ZDim					:= RequestPickingListFromHMI.Supportvert.ZDim;
			TFCalcoloFormaturaRT.Supporto.TipoPianoAppoggio 	:= 1;
			TFCalcoloFormaturaRT.Supporto.AltezzaDenteRitenuta	:= 20;
			TFCalcoloFormaturaRT.Supporto.ZDim_Ext1        	:= TFCalcoloFormaturaRT.Supporto.ZDim + TFCalcoloFormaturaRT.Supporto.AltezzaDenteRitenuta;
			TFCalcoloFormaturaRT.Supporto.DimBaseUtile		:= RequestPickingListFromHMI.Supportvert.DimBaseUtile;
			TFCalcoloFormaturaRT.Supporto.DimVertice 		:= RequestPickingListFromHMI.Supportvert.DimVertice*2;
			TFCalcoloFormaturaRT.Supporto.HMAX 				:= RequestPickingListFromHMI.Supportvert.HMAX;
			TFCalcoloFormaturaRT.Supporto.Tipologia 		:= BUNDLE;
			TFCalcoloFormaturaRT.Supporto.LatoDeposito 		:= 180;
			TFCalcoloFormaturaRT.TipoOrdinamento			:= 4;//Ordinamento di deposito, prima un lato poi l'altro
			TFCalcoloFormaturaRT.CalcolaFormatura := TRUE; 		//Lancio esecuzione dei calcoli
			MEMSET(ADR(FormaturaRT),0,SIZEOF(FormaturaRT));	//Pulisco la memoria di destinazione
			CalcolaFormaturaTrig2 := TRUE;
			TFCalcoloFormaturaRT.PulisciMemoria := FALSE;
		END_IF
	ELSIF (TFCalcoloFormaturaRT.CalcolaFormaturaDone OR TFCalcoloFormaturaRT.Errore > 0) AND CalcolaFormaturaTrig2 THEN
		TFCalcoloFormaturaRT.CalcolaFormatura := FALSE;
		FormaturaRT := TFCalcoloFormaturaRT.FormingSlab;
		CalcolaFormaturaTrig2 := FALSE;
		IF TFCalcoloFormaturaRT.Errore = 0 THEN
			CalcolaFormaturaTrig2 := FALSE;
			CalcolaFormingRT := FALSE;
		ELSE
			CalcolaFormingRT := TRUE;;
		END_IF
	END_IF
END_IF
TFCalcoloFormaturaRT();
END_ACTION

ACTION TEST_Variabili:

	Temp_Bool[8] := MachinePalletizer_TF.OUT.ClockSegnalazioni;
	Temp_Bool[9] := MachinePalletizer_TF.OUT.ClockSegnalazioniAlternato;

	Temp_Bool[0] := HMI_Status_BarrieraPall_OK;

  
 Temp_uint[0] := ElementiDaDepositare[1];	
 Temp_uint[0] := ElementiDaDepositare[2];		
 Temp_uint[0] := ElementiDaDepositare[3];
		 
 Temp_uint[0] := HMI_WorkAreaDataPicking[1].NumElementiDaLavorare;	
 Temp_uint[0] := HMI_WorkAreaDataPicking[1].NumElementiDaLavorare;		

	
 Temp_Real[1]:= 	MachinePalletizer_TF.WorkSpace[1].X;
 Temp_Real[1]:= 	MachinePalletizer_TF.WorkSpace[1].Y;
 Temp_Real[1]:= 	MachinePalletizer_TF.WorkSpace[1].Z;
   
 
 Temp_Real[1]:= Traiettoria.StartPoint.X;
 Temp_Real[1]:= Traiettoria.StartPoint.Y;
 Temp_Real[1]:= Traiettoria.StartPoint.Z;
 Temp_Real[1]:= Traiettoria.StartPoint.J;


//; SimulazioneSenzaPalletFalde;
//PINZA
Temp_Real[1]:= Pinza.Ovem1.Status.ValoreDepressioneIstantanea;
Temp_Real[1]:= HMI_DepressioneOVEM_DX1;
Temp_Real[1]:= Pinza.Ovem12.Status.ValoreDepressioneIstantanea;
Temp_Real[1]:= HMI_DepressioneOVEM_DX2;
//;
Temp_Real[1]:= Pinza.Ovem22.Status.ValoreDepressioneIstantanea;
Temp_Real[1]:= HMI_DepressioneOVEM_SX1;
Temp_Real[1]:= Pinza.Ovem22.Status.ValoreDepressioneIstantanea;
Temp_Real[1]:= HMI_DepressioneOVEM_SX2;
	
//Presenza
//FormaturaAFRAMERT;
Temp_bool[0] := I_PresenzaSupporto[1];
Temp_bool[0] := I_PresenzaBundle[1];
Temp_bool[0] := I_PresenzaCentrale[1];
Temp_bool[0] := I_PHPresenzaPallet[1];
Temp_bool[0] := I_PHPresenzaPalletVirtuale[1];

Temp_bool[0] := I_PresenzaSupporto[2];
Temp_bool[0] := I_PresenzaBundle[2];
Temp_bool[0] := I_PresenzaCentrale[2];
Temp_bool[0] := I_PHPresenzaPallet[2];
Temp_bool[0] := I_PHPresenzaPalletVirtuale[2];

Temp_bool[0] := I_PresenzaSupporto[3];
Temp_bool[0] := I_PresenzaBundle[3];
Temp_bool[0] := I_PresenzaCentrale[3];
Temp_bool[0] := I_PHPresenzaPallet[3];
Temp_bool[0] := I_PHPresenzaPalletVirtuale[3];

//*** Calcola Lista produzione  ***	

 Temp_bool[0] := HMI_WorkAreaDataPicking[1].Destinazione; // (0=Prelievo, 1= deposito).	
 Temp_bool[0] := HMI_WorkAreaDataPicking[2].Destinazione;
 Temp_bool[0] := HMI_WorkAreaDataPicking[3].Destinazione;
 Temp_bool[0] := HMI_WorkAreaDataPicking[4].Destinazione;
 
//valori dei supporti della lista 2
Temp_Real[1]:= RequestPickingListFromHMI[2].SupportPianoLegno.XDim;
Temp_Real[1]:= RequestPickingListFromHMI[2].SupportPianoLegno.YDim;	
Temp_real[1]:= RequestPickingListFromHMI[2].SupportPianoLegno.ZDim;
Temp_INT[0]	:= RequestPickingListFromHMI[2].State; 						//Stato WO richiesto
Temp_UINT[0]:= RequestPickingListFromHMI[2].SlabNumber;			// Numero Lastre da depositare

// compilazione WO
// Tipologia: 0= Orrizzontale LEGNO,1= Orrizzontale Telaio , 2 = Bundle, 3 = A-FRAME
Temp_INT[0] := WorkareaState[1].Supporto.Tipologia;
Temp_INT[0] := WorkareaState[2].Supporto.Tipologia;
Temp_INT[0] := WorkareaState[3].Supporto.Tipologia;
Temp_INT[0] := WorkareaState[4].Supporto.Tipologia;
	//...	
Temp_INT[0] := WorkareaState[8].Supporto.Tipologia;

IF (FALSE) THEN
(*
// Per ogni Postazione
// Postazione 1	
//	HMI_WorkAreaDataPicking[1].Destinazione := 0;		//Prel/Depo
	HMI_WorkAreaDataPicking[1].Typology := 0;			//Cassa,Telaio,...
	HMI_WorkAreaDataPicking[1].NumElementiDaLavorare := 0; // Lastre da prelevare, se la Postazione è di deposito, SCOMPARE!
	HMI_NumeroLastreRimanentiOrdineAttuale[1] :=0;	
	HMI_WorkAreaDataPicking[1].NumElementiDaLavorare := 0; // dopo la Barra
	HMI_NumeroPezziPresentiPostazione[1] :=0;			//Campo sotto la cornice	
// Postazione 2	
	HMI_WorkAreaDataPicking[2].Destinazione := 0;		//Prel/Depo
	HMI_WorkAreaDataPicking[2].Typology := 0;			//Cassa,Telaio,...
	HMI_WorkAreaDataPicking[2].NumElementiDaLavorare := 0; // Lastre da prelevare, se la Postazione è di deposito, SCOMPARE!
	HMI_NumeroLastreRimanentiOrdineAttuale[2] :=0;	
	HMI_WorkAreaDataPicking[2].NumElementiDaLavorare := 0; // dopo la Barra
	HMI_NumeroPezziPresentiPostazione[2] :=0;			//Campo sotto la cornice	
// Postazione 3
	HMI_WorkAreaDataPicking[3].Destinazione := 0;		//Prel/Depo
	HMI_WorkAreaDataPicking[3].Typology := 0;			//Cassa,Telaio,...
	HMI_WorkAreaDataPicking[3].NumElementiDaLavorare := 0; // Lastre da prelevare, se la Postazione è di deposito, SCOMPARE!
	HMI_NumeroLastreRimanentiOrdineAttuale[3] :=0;
	HMI_WorkAreaDataPicking[3].NumElementiDaLavorare := 0; // dopo la Barra
	HMI_NumeroPezziPresentiPostazione[3] :=0;			//Campo sotto la cornice	


// Work Order Richiesto
	RequestPickingListFromHMI[2].State :=0;
	RequestPickingListFromHMI[2].SlabNumber :=0;
// Work Order attuale	
	ActualPickingListFromHMI[2].State  :=0;	
	HMI_NumeroLastreDepOrdineAttuale[2] :=0; 
	RequestPickingListFromHMI[2].SlabNumber :=0;
	
	ElementiDaDepositare[Temp_IdxLista]  := Temp_UINT[0]; //# Somma delle Lastre da Prelevare nelle WorkArea
	WorkAreaState[Temp_i].P := Temp_INT[0];				//# Pack Poinyer, contiene il NumElementiDaLavorare
	
	//Controllo sul numero elementi da prelevare che deve essere min o uguale agli elementi da depositare
	ActualPickingListFromHMI[Temp_IdxLista]	:= RequestPickingListFromHMI[Temp_IdxLista];
	ActualPickingListFromHMI[Temp_IdxLista].State 	:= e_StatoWorkOrder.DA_ESEGUIRE;
	
	Temp_INT[0] := Picking.RequestPickingListFromHMI[1].SupportPianoLegno.Code;
	Temp_INT[0]	:= RequestPickingListFromHMI[Temp_IdxLista].SupportPianoLegno.Code;
	Temp_REAL[0] := RequestPickingListFromHMI[Temp_IdxLista].SupportPianoLegno.XDim;
	Temp_REAL[0] := RequestPickingListFromHMI[Temp_IdxLista].SupportPianoLegno.YDim;
	Temp_REAL[0] := RequestPickingListFromHMI[Temp_IdxLista].SupportPianoLegno.ZDim;
	Temp_INT[3] := HMI_WorkAreaDataPicking[1].Typology;

	// Lista di produzione compilata
	//WorkAreaProductionList[MAXAREA].PElementList[MAXELEMENTLIST].WA_PRELIEVO :=0;
	//WorkAreaProductionList[MAXAREA].PElementList[MAXELEMENTLIST].WA_DEPOSITO :=0;
	
	//Work Area Production List 1
	WorkAreaProductionList[1].PElementList[1].WA_PRELIEVO :=0;
	WorkAreaProductionList[1].PElementList[2].WA_PRELIEVO :=0;
	WorkAreaProductionList[1].PElementList[3].WA_PRELIEVO :=0;
	
	WorkAreaProductionList[1].PElementList[1].WA_DEPOSITO :=0;
	WorkAreaProductionList[1].PElementList[2].WA_DEPOSITO :=0;
	WorkAreaProductionList[1].PElementList[3].WA_DEPOSITO :=0;
	//Work Area Production List 2	
	WorkAreaProductionList[2].PElementList[1].WA_PRELIEVO :=0;
	WorkAreaProductionList[2].PElementList[2].WA_PRELIEVO :=0;
	WorkAreaProductionList[2].PElementList[3].WA_PRELIEVO :=0;
	WorkAreaProductionList[2].PElementList[4].WA_PRELIEVO :=0;
	WorkAreaProductionList[2].PElementList[5].WA_PRELIEVO :=0;
		
	WorkAreaProductionList[2].PElementList[1].WA_DEPOSITO :=0;
	WorkAreaProductionList[2].PElementList[2].WA_DEPOSITO :=0;
	WorkAreaProductionList[2].PElementList[3].WA_DEPOSITO :=0;
	WorkAreaProductionList[2].PElementList[4].WA_DEPOSITO :=0;
	WorkAreaProductionList[2].PElementList[5].WA_DEPOSITO :=0;
//Work Area Production List 3 (WA dove viene fatto il prelievo con 5 lastre da spostare)
	WorkAreaProductionList[3].PElementList[1].WA_PRELIEVO :=0;
	WorkAreaProductionList[3].PElementList[2].WA_PRELIEVO :=0;
	WorkAreaProductionList[3].PElementList[3].WA_PRELIEVO :=0;
	WorkAreaProductionList[3].PElementList[4].WA_PRELIEVO :=0;
	WorkAreaProductionList[3].PElementList[5].WA_PRELIEVO :=0;
	WorkAreaProductionList[3].PElementList[6].WA_PRELIEVO :=0;
							 //(WA dove viene fatto il deposito con 5 lastre da spostare)
	WorkAreaProductionList[3].PElementList[1].WA_DEPOSITO :=0;
	WorkAreaProductionList[3].PElementList[2].WA_DEPOSITO :=0;
	WorkAreaProductionList[3].PElementList[3].WA_DEPOSITO :=0;
	WorkAreaProductionList[3].PElementList[4].WA_DEPOSITO :=0;
	WorkAreaProductionList[3].PElementList[5].WA_DEPOSITO :=0;
	WorkAreaProductionList[3].PElementList[6].WA_DEPOSITO :=0;
//Work Area Production List 4
	WorkAreaProductionList[4].PElementList[1].WA_PRELIEVO :=0;
	WorkAreaProductionList[4].PElementList[2].WA_PRELIEVO :=0;
	WorkAreaProductionList[4].PElementList[3].WA_PRELIEVO :=0;
	WorkAreaProductionList[4].PElementList[4].WA_PRELIEVO :=0;
	WorkAreaProductionList[4].PElementList[5].WA_PRELIEVO :=0;
		
	WorkAreaProductionList[4].PElementList[1].WA_DEPOSITO :=0;
	WorkAreaProductionList[4].PElementList[2].WA_DEPOSITO :=0;
	WorkAreaProductionList[4].PElementList[3].WA_DEPOSITO :=0;
	WorkAreaProductionList[4].PElementList[4].WA_DEPOSITO :=0;
	WorkAreaProductionList[4].PElementList[5].WA_DEPOSITO :=0;	
	
// TEST SE LISTA E' ATTIVATA
	ActualPickingListFromHMI[1].State :=0;//Ordine postazioni 1..8 in lavoro
	ActualPickingListFromHMI[2].State :=0;//Ordine postazioni 1..4 in lavoro
	ActualPickingListFromHMI[3].State :=0;//Ordine postazioni 5..8 in lavoro
		
	HMI_WorkAreaDataPicking_1_8 := 0;//Ordine postazioni 1..8 in lavoro
	HMI_WorkAreaDataPicking_1_4 := 0;//Ordine postazioni 1..4 in lavoro
	HMI_WorkAreaDataPicking_5_8 := 0;//Ordine postazioni 5..8 in lavoro
*)	
END_IF
END_ACTION

END_PROGRAM

// ---- POUs/TFPalletizerData_Lastre/TFPalletizerGestione_PickPoint_Rulliere.TcPOU
FUNCTION_BLOCK TFPalletizerGestione_PickPoint_Rulliere
(* Valorizza e aggiorna le variabili di stato del Pick-Point sulla base dei valori ricevuti dalla linea e dai valori inviati alla linea *)
VAR_INPUT
	WorkPickPoint : POINTER TO ARRAY [1..MAXPICKPOINT] OF TFMachinePalletizer_WorkPickPointSlab;
	WorkPickPointState : POINTER TO ARRAY [1..MAXPICKPOINT] OF TFMachinePalletizer_WorkPickPoint_State;
	WorkPickPointStateDaLinea : POINTER TO ARRAY [1..MAXPICKPOINT] OF TFMachinePalletizer_WorkPickPointRoller_State_DaLinea;
	WorkPickPointStateALinea : POINTER TO ARRAY [1..MAXPICKPOINT] OF TFMachinePalletizer_WorkPickPointRoller_State_ALinea;

END_VAR
VAR_OUTPUT
END_VAR
VAR
	wpp : INT;
END_VAR


FOR wpp:= 1 TO MAXPICKPOINT DO 
(******************* Valorizzazione da LINEA a PALLETTIZZATORE *********************)
	(* Set stato *)
	IF WorkPickPointStateDaLinea^[wpp].Automatico THEN
		WorkPickPointState^[wpp].State := WORKPICKPOINT_STATE_AUTO;
	ELSIF NOT WorkPickPointStateDaLinea^[wpp].Automatico THEN
		WorkPickPointState^[wpp].State := WORKPICKPOINT_STATE_MAN;
	ELSIF WorkPickPointStateDaLinea^[wpp].Errore THEN
		WorkPickPointState^[wpp].State := WORKPICKPOINT_STATE_ERROR;
	END_IF
	(* Set Marcia Presente/Assente *)
	IF WorkPickPointStateDaLinea^[wpp].PowerOK THEN
		WorkPickPointState^[wpp].PowerOK := TRUE;
	ELSE
		WorkPickPointState^[wpp].PowerOK := FALSE;
	END_IF
	(* Set Lastra Presente/Assente *)
	IF WorkPickPointStateDaLinea^[wpp].Occupato THEN
		WorkPickPointState^[wpp].ProdPresence := PROD_PRESENTE;
	ELSE
		WorkPickPointState^[wpp].ProdPresence := PROD_ASSENTE;
	END_IF
	(* Set Lastra Pronta/Non Pronta *)
	IF WorkPickPointStateDaLinea^[wpp].LastraPronta THEN
		WorkPickPointState^[wpp].LastraPronta := TRUE;
	ELSE
		WorkPickPointState^[wpp].LastraPronta := FALSE;
	END_IF
	(* Set CODICE *)
	WorkPickPointState^[wpp].Code := WorkPickPointStateDaLinea^[wpp].Codice; 
	(* Set Priorità *)
	IF WorkPickPointStateDaLinea^[wpp].Priority THEN
		WorkPickPointState^[wpp].Priority := MAX_PRIORITY;
	ELSE
		WorkPickPointState^[wpp].Priority := Min_PRIORITY;
	END_IF
	
(******************* Valorizzazione da PALLETTIZZATORE a LINEA *********************)	
	(* Set stato ingombro *)
	IF WorkPickPointState^[wpp].StatoIngombroEE = EE_IN_INGOMBRO THEN
		WorkPickPointStateALinea^[wpp].Ingombro 	:= TRUE;
	ELSIF WorkPickPointState^[wpp].StatoIngombroEE 	 = EE_FUORI_INGOMBRO THEN
		WorkPickPointStateALinea^[wpp].Ingombro 	:= FALSE;
	END_IF
	(* Set stato Prelievo *)
	IF WorkPickPointState^[wpp].StatoPrelievo = PRELIEVO_DA_EFFETTUARE THEN
		WorkPickPointStateALinea^[wpp].Prelievo_Effettuato := FALSE;
	ELSIF WorkPickPointState^[wpp].StatoPrelievo = PRELIEVO_EFFETTUATO THEN
		WorkPickPointStateALinea^[wpp].Prelievo_Effettuato := TRUE;
	END_IF

END_FOR

END_FUNCTION_BLOCK

// ---- POUs/TFPalletizerData_Lastre/TFAggiuntaSupportoManuale.TcPOU
FUNCTION_BLOCK TFAggiuntaSupportoManuale
VAR_INPUT
	WorkArea : POINTER TO ARRAY [1..MAXAREA] OF TFMachinePalletizer_WorkArea;
	WorkAreaState : POINTER TO ARRAY [1..MAXAREA] OF TFMachinePalletizer_WorkAreaState;
	WorkAreaNumber : UINT; //Numero postazione
	Forming : POINTER TO ARRAY [1..MAXFORMING] OF TFMachinePalletizer_FormingForSlab;
	Pallet : POINTER TO ARRAY [1..MAXPALLET] OF TFMachinePalletizer_Pallet;
	Layer : POINTER TO ARRAY [1..MAXLAYER] OF TFMachinePalletizer_Layer;
	ProgressiveNrWA : POINTER TO UDINT;
	CodicePostazione : INT;
	IndiceFormaturaPostazione : INT;
	AbilitaAssegnazioneCodicePiazzoleConPaccoSuRibaltino : BOOL;
	InserisciNuovoPallet : BOOL;
	PH_Presenza : bool;// ARRAY[1..MAXAREA] OF BOOL;
END_VAR
VAR_OUTPUT
END_VAR
VAR
	PHPostazioniUPTrig 			: ARRAY[1..MAXAREA] OF BOOL;
	PHPostazioniDOWNTrig 		: ARRAY[1..MAXAREA] OF BOOL;
	UltimaFormaturaAssegnata 	: INT;
	UltimaPostazioneCancellata 	: UINT;
	UltimaPostazioneCreata 		: UINT;
	Zone : INT;
	ar: INT;
	cod : INT;
	FormaturaZona : ARRAY[1..MAXFORMINGCODE] OF INT;
	FormaturePresenti : ARRAY[1..MAXFORMING] OF INT;
	DoppiaFormaturaAttiva :BOOL;
	CodiceInFormaturaMem : INT;
	NumCodiciInFormaturaAttiviPerZona : UINT;	

END_VAR

InserisciNuovoPallet:= FALSE;
//Fronte salita
IF PH_Presenza AND NOT PHPostazioniUPTrig[WorkAreaNumber] THEN
	PHPostazioniUPTrig[WorkAreaNumber] := TRUE;
	UltimaPostazioneCreata := WorkAreaNumber;
ELSIF NOT PH_Presenza AND PHPostazioniUPTrig[WorkAreaNumber] THEN
	PHPostazioniUPTrig[WorkAreaNumber] := FALSE;
END_IF
//Fronte discesa
//Pulisco la postazione
IF NOT PH_Presenza AND NOT PHPostazioniDOWNTrig[WorkAreaNumber] THEN
	PHPostazioniDOWNTrig[WorkAreaNumber] := TRUE;
	UltimaPostazioneCancellata := WorkAreaNumber;
	IF WorkAreaState^[WorkAreaNumber].State >= WORKAREA_STATE_OCCUPIED_WORKING THEN
		TFClearWorkAreaArray(WorkArea,WorkAreaState,WorkAreaNumber);
	END_IF
	
	IF WorkAreaNumber = Mission.PPlace THEN
	//Modificacion borrar datos piking Al sacar el soporte
	MEMSET(destAddr := ADR(HMi_DimensionesPiezasWorkAreaDeposito),fillByte := 0 , n := SIZEOF(HMi_DimensionesPiezasWorkAreaDeposito));
	END_IF
	
ELSIF PH_Presenza AND PHPostazioniDOWNTrig[WorkAreaNumber] THEN
	PHPostazioniDOWNTrig[WorkAreaNumber] := FALSE;
END_IF

//Verifico se è stato inserito il nuovo codice del pallet
IF (WorkAreaState^[WorkAreaNumber].Code > 0 OR PHPostazioniUPTrig[WorkAreaNumber]) AND (WorkArea^[WorkAreaNumber].Enable = 1 AND WorkAreaState^[WorkAreaNumber].State < WORKAREA_STATE_OCCUPIED_WORKING AND WorkAreaState^[WorkAreaNumber].State <> 1) THEN
	InserisciNuovoPallet := TRUE;
END_IF

IF InserisciNuovoPallet AND WorkAreaState^[WorkAreaNumber].State < WORKAREA_STATE_OCCUPIED_WORKING THEN	
	
	WorkAreaState^[WorkAreaNumber].Taped := -1;
	WorkAreaState^[WorkAreaNumber].LGV_ReqAbort := FALSE;
	
